KUKA KRL program: ps_b_ltb_res_c02.src, ps_b_ltb_res_c02.dat

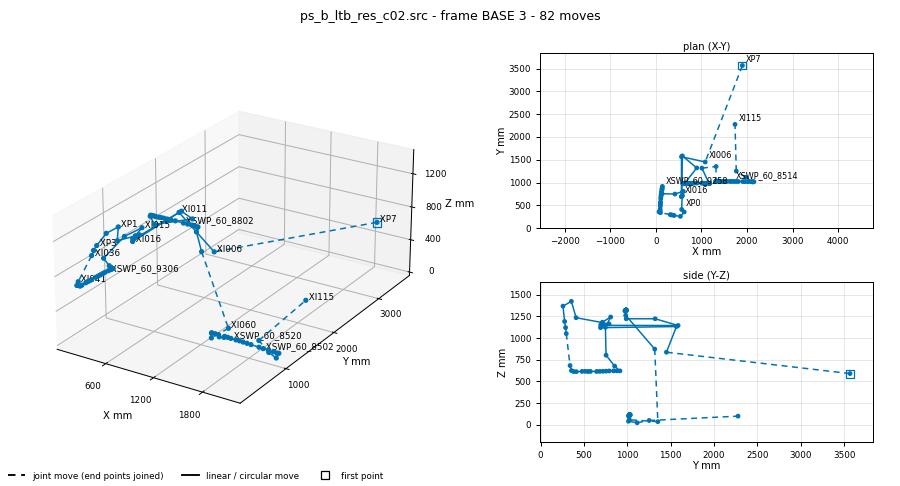
[picture p0: tool path of ps_b_ltb_res_c02.src in frame BASE 3, 82 of 82 moves have a stored position in this frame; points joined in program order, loops and branches not executed]
--- ps_b_ltb_res_c02.src ---
&ACCESS RVO1
&COMMENT Solda Axor LTB
&PARAM DISKPATH = KRC:\R1\Program\OLP
DEF ps_b_ltb_res_c02( )
;FOLD INI
;FOLD SPOTTECH INI
USERSPOT(#INIT)
;ENDFOLD (SPOTTECH INI)
;FOLD GRIPPERTECH INI
USER_GRP(0,DUMMY,DUMMY,GDEFAULT)
;ENDFOLD (GRIPPERTECH INI)
  ;FOLD USER INI
    ;Make your modifications here

  ;ENDFOLD (USER INI)
;ENDFOLD (INI)

; Caracterizacao dos meios de producao
; Changes: Solda Respot - AXOR - LTB
; Versao Atual: 26/03/2016
; Ferramenta : Gun C02
; Name: P13.060-R2

chk_w3_wechs_ok ( )     ; CHECK GUN C2

IF (NOT(GHOST())) THEN
IF MaxStandMenge(3) THEN
  MaxStandmengeErreicht(3)
ENDIF
IF Elektrodenwechsel(3) THEN
  e_Fraes3 ()
ENDIF
ENDIF

;FOLD PTP P7 Vel=100 % PDAT2 Tool[4]:Gun C03 Base[3]:Atego/Axor;%{PE}%R 8.2.20,%MKUKATPBASIS,%CMOVE,%VPTP,%P 1:PTP, 2:P7, 3:, 5:100, 7:PDAT2
$BWDSTART=FALSE
PDAT_ACT=PPDAT2
FDAT_ACT=FP7
BAS(#PTP_PARAMS,100)
PTP XP7
;ENDFOLD

;FOLD OUT 3380 'Perfil Livre Estacao' State=TRUE ;%{PE}%R 8.2.20,%MKUKATPBASIS,%COUT,%VOUTX,%P 2:3380, 3:Perfil Livre Estacao, 5:TRUE, 6:
$OUT[3380]=TRUE
;ENDFOLD
;FOLD WAIT FOR ( IN 3380 'Liberacao de Solda' );%{PE}%R 8.2.20,%MKUKATPBASIS,%CEXT_WAIT_FOR,%VEXT_WAIT_FOR,%P 2:, 4:, 5:$IN, 6:3380, 7:Liberacao de Solda, 9:
WAIT FOR  ( $IN[3380] )
;ENDFOLD
;FOLD OUT 3380 'Perfil Livre Estacao' State=FALSE ;%{PE}%R 8.2.20,%MKUKATPBASIS,%COUT,%VOUTX,%P 2:3380, 3:Perfil Livre Estacao, 5:FALSE, 6:
$OUT[3380]=FALSE
;ENDFOLD

;FOLD ; Liga intertravamento 3 c/ R03;%{PE}%R 8.2.20,%MKUKATPBASIS,%CCOMMENT,%VNORMAL,%P 2:Liga  intertravamento 3 c/  R03
;ENDFOLD
;FOLD Collision.Monitoring_3_On ;%{PE}%MKUKATPUSER
COLLSTOP( 3, 1 ) ;Interrupt-Controlled
;ENDFOLD

;FOLD ; Liga intertravamento 10 c/ R04;%{PE}%R 8.2.20,%MKUKATPBASIS,%CCOMMENT,%VNORMAL,%P 2:Liga  intertravamento 10 c/  R04
;ENDFOLD
;FOLD Collision.Monitoring_10_On ;%{PE}%MKUKATPUSER
COLLSTOP( 10, 1 ) ;not Interrupt-Controlled
;ENDFOLD
;FOLD ; ;%{PE}%R 8.2.20,%MKUKATPBASIS,%CCOMMENT,%VNORMAL,%P 2:
;ENDFOLD
;FOLD ; Liga intertravamento 5 c/ R05;%{PE}%R 8.2.20,%MKUKATPBASIS,%CCOMMENT,%VNORMAL,%P 2:Liga  intertravamento 5 c/  R05
;ENDFOLD
;FOLD Collision.Monitoring_5_On ;%{PE}%MKUKATPUSER
COLLSTOP( 5, 1 ) ;not Interrupt-Controlled
;ENDFOLD

;FOLD ; Liga intertravamento 9 c/ R05;%{PE}%R 8.2.20,%MKUKATPBASIS,%CCOMMENT,%VNORMAL,%P 2:Liga  intertravamento 9 c/  R05
;ENDFOLD
;FOLD Collision.Monitoring_9_On ;%{PE}%MKUKATPUSER
COLLSTOP( 9, 1 ) ;not Interrupt-Controlled
;ENDFOLD

;FOLD ; Liga intertravamento 14 c/ R05;%{PE}%R 8.2.20,%MKUKATPBASIS,%CCOMMENT,%VNORMAL,%P 2:Liga  intertravamento 14 c/  R05
;ENDFOLD
;FOLD Collision.Monitoring_14_On ;%{PE}%MKUKATPUSER
COLLSTOP( 14, 1 ) ;not Interrupt-Controlled
;ENDFOLD
;FOLD ; ;%{PE}%R 8.2.20,%MKUKATPBASIS,%CCOMMENT,%VNORMAL,%P 2:
;ENDFOLD
;FOLD PTP l006 CONT Vel=100 % P_OLP4 Tool[3]:Pinca C2 Base[3]:Atego/Axor;%{PE}%R 8.2.20,%MKUKATPBASIS,%CMOVE,%VPTP,%P 1:PTP, 2:l006, 3:C_DIS, 5:100, 7:P_OLP4
$BWDSTART=FALSE
PDAT_ACT=PP_OLP4
FDAT_ACT=Fl006
BAS(#PTP_PARAMS,100)
PTP Xl006 C_DIS
;ENDFOLD
;FOLD LIN l011 CONT Vel=2 m/s L_OLP48 Tool[3]:Pinca C2 Base[3]:Atego/Axor;%{PE}%R 8.2.20,%MKUKATPBASIS,%CMOVE,%VLIN,%P 1:LIN, 2:l011, 3:C_DIS C_DIS, 5:2, 7:L_OLP48
$BWDSTART=FALSE
LDAT_ACT=LL_OLP48
FDAT_ACT=Fl011
BAS(#CP_PARAMS,2)
LIN Xl011 C_DIS C_DIS
;ENDFOLD
;FOLD LIN l016 CONT Vel=2 m/s L_OLP49 Tool[3]:Pinca C2 Base[3]:Atego/Axor;%{PE}%R 8.2.20,%MKUKATPBASIS,%CMOVE,%VLIN,%P 1:LIN, 2:l016, 3:C_DIS C_DIS, 5:2, 7:L_OLP49
$BWDSTART=FALSE
LDAT_ACT=LL_OLP49
FDAT_ACT=Fl016
BAS(#CP_PARAMS,2)
LIN Xl016 C_DIS C_DIS
;ENDFOLD
;FOLD PTP l021 CONT Vel=100 % P_OLP5 Tool[3]:Pinca C2 Base[3]:Atego/Axor;%{PE}%R 8.2.20,%MKUKATPBASIS,%CMOVE,%VPTP,%P 1:PTP, 2:l021, 3:C_DIS, 5:100, 7:P_OLP5
$BWDSTART=FALSE
PDAT_ACT=PP_OLP5
FDAT_ACT=Fl021
BAS(#PTP_PARAMS,100)
PTP Xl021 C_DIS
;ENDFOLD
;FOLD LIN l026 CONT Vel=2 m/s L_OLP50 Tool[3]:Pinca C2 Base[3]:Atego/Axor;%{PE}%R 8.2.20,%MKUKATPBASIS,%CMOVE,%VLIN,%P 1:LIN, 2:l026, 3:C_DIS C_DIS, 5:2, 7:L_OLP50
$BWDSTART=FALSE
LDAT_ACT=LL_OLP50
FDAT_ACT=Fl026
BAS(#CP_PARAMS,2)
LIN Xl026 C_DIS C_DIS
;ENDFOLD
;FOLD LIN P0 CONT Vel=2 m/s CPDAT0 Tool[3]:Pinca C2 Base[3]:Atego/Axor;%{PE}%R 8.2.20,%MKUKATPBASIS,%CMOVE,%VLIN,%P 1:LIN, 2:P0, 3:C_DIS C_DIS, 5:2, 7:CPDAT0
$BWDSTART=FALSE
LDAT_ACT=LCPDAT0
FDAT_ACT=FP0
BAS(#CP_PARAMS,2)
LIN XP0 C_DIS C_DIS
;ENDFOLD
;FOLD LIN P1 CONT Vel=2 m/s CPDAT1 Tool[3]:Pinca C2 Base[3]:Atego/Axor;%{PE}%R 8.2.20,%MKUKATPBASIS,%CMOVE,%VLIN,%P 1:LIN, 2:P1, 3:C_DIS C_DIS, 5:2, 7:CPDAT1
$BWDSTART=FALSE
LDAT_ACT=LCPDAT1
FDAT_ACT=FP1
BAS(#CP_PARAMS,2)
LIN XP1 C_DIS C_DIS
;ENDFOLD
;FOLD LIN P2 CONT Vel=2 m/s CPDAT2 Tool[3]:Pinca C2 Base[3]:Atego/Axor;%{PE}%R 8.2.20,%MKUKATPBASIS,%CMOVE,%VLIN,%P 1:LIN, 2:P2, 3:C_DIS C_DIS, 5:2, 7:CPDAT2
$BWDSTART=FALSE
LDAT_ACT=LCPDAT2
FDAT_ACT=FP2
BAS(#CP_PARAMS,2)
LIN XP2 C_DIS C_DIS
;ENDFOLD
;FOLD LIN P3 CONT Vel=2 m/s CPDAT3 Tool[3]:Pinca C2 Base[3]:Atego/Axor;%{PE}%R 8.2.20,%MKUKATPBASIS,%CMOVE,%VLIN,%P 1:LIN, 2:P3, 3:C_DIS C_DIS, 5:2, 7:CPDAT3
$BWDSTART=FALSE
LDAT_ACT=LCPDAT3
FDAT_ACT=FP3
BAS(#CP_PARAMS,2)
LIN XP3 C_DIS C_DIS
;ENDFOLD
;FOLD LIN l031 CONT Vel=2 m/s L_OLP51 Tool[3]:Pinca C2 Base[3]:Atego/Axor;%{PE}%R 8.2.20,%MKUKATPBASIS,%CMOVE,%VLIN,%P 1:LIN, 2:l031, 3:C_DIS C_DIS, 5:2, 7:L_OLP51
$BWDSTART=FALSE
LDAT_ACT=LL_OLP51
FDAT_ACT=Fl031
BAS(#CP_PARAMS,2)
LIN Xl031 C_DIS C_DIS
;ENDFOLD
;FOLD PTP l036 CONT Vel=100 % P_OLP6 Tool[3]:Pinca C2 Base[3]:Atego/Axor;%{PE}%R 8.2.20,%MKUKATPBASIS,%CMOVE,%VPTP,%P 1:PTP, 2:l036, 3:C_DIS, 5:100, 7:P_OLP6
$BWDSTART=FALSE
PDAT_ACT=PP_OLP6
FDAT_ACT=Fl036
BAS(#PTP_PARAMS,100)
PTP Xl036 C_DIS
;ENDFOLD
;FOLD PTP l041 CONT Vel=100 % P_OLP7 Tool[3]:Pinca C2 Base[3]:Atego/Axor;%{PE}%R 8.2.20,%MKUKATPBASIS,%CMOVE,%VPTP,%P 1:PTP, 2:l041, 3:C_DIS, 5:100, 7:P_OLP7
$BWDSTART=FALSE
PDAT_ACT=PP_OLP7
FDAT_ACT=Fl041
BAS(#PTP_PARAMS,100)
PTP Xl041 C_DIS
;ENDFOLD
;FOLD LIN l046 CONT Vel=2 m/s L_OLP52 Tool[3]:Pinca C2 Base[3]:Atego/Axor;%{PE}%R 8.2.20,%MKUKATPBASIS,%CMOVE,%VLIN,%P 1:LIN, 2:l046, 3:C_DIS C_DIS, 5:2, 7:L_OLP52
$BWDSTART=FALSE
LDAT_ACT=LL_OLP52
FDAT_ACT=Fl046
BAS(#CP_PARAMS,2)
LIN Xl046 C_DIS C_DIS
;ENDFOLD

;FOLD ; SWP_60_9280;%{PE}%R 8.2.20,%MKUKATPBASIS,%CCOMMENT,%VNORMAL,%P 2:SWP_60_9280
;ENDFOLD
;FOLD LIN SWP_60_9280 L_OLP53 SPOT Gun=2 RETR CLS PgNo1=186 ACTIVE=1 NORMAL Tool[3]:Pinca C2 Base[3]:Atego/Axor;%{PE}%R 8.2.2,%MKUKATPSPOT,%CSPOT,%VLIN,%P 1:LIN, 2:SWP_60_9280, 3:, 5:2, 7:L_OLP53, 10:2, 12:#FIRST, 14:#CLO, 16:186, 18:1, 20:0, 22:0, 24:1, 25:NORMAL
$BWDSTART=FALSE
LDAT_ACT=LL_OLP53
FDAT_ACT=FSWP_60_9280
BAS(#CP_PARAMS,LL_OLP53.VEL)
S_ACT.GUN=2
S_ACT.PAIR=SDEFAULT.PAIR
S_ACT.RETR=#CLO
S_ACT.CLO_TM=1
S_ACT.PGNO1=186
S_ACT.PGNO2=SDEFAULT.PGNO2
S_ACT.PRESS1=SDEFAULT.PRESS1
S_ACT.PRESS2=SDEFAULT.PRESS2
S_READY=FALSE
LIN XSWP_60_9280
USERSPOT(#SPOT, S_ACT)
WAIT FOR S_READY
;ENDFOLD

;FOLD ; SWP_60_9282;%{PE}%R 8.2.20,%MKUKATPBASIS,%CCOMMENT,%VNORMAL,%P 2:SWP_60_9282
;ENDFOLD
;FOLD LIN SWP_60_9282 L_OLP54 SPOT Gun=2 RETR CLS PgNo1=186 ACTIVE=1 NORMAL Tool[3]:Pinca C2 Base[3]:Atego/Axor;%{PE}%R 8.2.2,%MKUKATPSPOT,%CSPOT,%VLIN,%P 1:LIN, 2:SWP_60_9282, 3:, 5:2, 7:L_OLP54, 10:2, 12:#FIRST, 14:#CLO, 16:186, 18:1, 20:0, 22:0, 24:1, 25:NORMAL
$BWDSTART=FALSE
LDAT_ACT=LL_OLP54
FDAT_ACT=FSWP_60_9282
BAS(#CP_PARAMS,LL_OLP54.VEL)
S_ACT.GUN=2
S_ACT.PAIR=SDEFAULT.PAIR
S_ACT.RETR=#CLO
S_ACT.CLO_TM=1
S_ACT.PGNO1=186
S_ACT.PGNO2=SDEFAULT.PGNO2
S_ACT.PRESS1=SDEFAULT.PRESS1
S_ACT.PRESS2=SDEFAULT.PRESS2
S_READY=FALSE
LIN XSWP_60_9282
USERSPOT(#SPOT, S_ACT)
WAIT FOR S_READY
;ENDFOLD

;FOLD ; SWP_60_9286;%{PE}%R 8.2.20,%MKUKATPBASIS,%CCOMMENT,%VNORMAL,%P 2:SWP_60_9286
;ENDFOLD
;FOLD LIN SWP_60_9286 L_OLP55 SPOT Gun=2 RETR CLS PgNo1=186 ACTIVE=1 NORMAL Tool[3]:Pinca C2 Base[3]:Atego/Axor;%{PE}%R 8.2.2,%MKUKATPSPOT,%CSPOT,%VLIN,%P 1:LIN, 2:SWP_60_9286, 3:, 5:2, 7:L_OLP55, 10:2, 12:#FIRST, 14:#CLO, 16:186, 18:1, 20:0, 22:0, 24:1, 25:NORMAL
$BWDSTART=FALSE
LDAT_ACT=LL_OLP55
FDAT_ACT=FSWP_60_9286
BAS(#CP_PARAMS,LL_OLP55.VEL)
S_ACT.GUN=2
S_ACT.PAIR=SDEFAULT.PAIR
S_ACT.RETR=#CLO
S_ACT.CLO_TM=1
S_ACT.PGNO1=186
S_ACT.PGNO2=SDEFAULT.PGNO2
S_ACT.PRESS1=SDEFAULT.PRESS1
S_ACT.PRESS2=SDEFAULT.PRESS2
S_READY=FALSE
LIN XSWP_60_9286
USERSPOT(#SPOT, S_ACT)
WAIT FOR S_READY
;ENDFOLD

;FOLD ; SWP_60_9288;%{PE}%R 8.2.20,%MKUKATPBASIS,%CCOMMENT,%VNORMAL,%P 2:SWP_60_9288
;ENDFOLD
;FOLD LIN SWP_60_9288 L_OLP56 SPOT Gun=2 RETR CLS PgNo1=186 ACTIVE=1 NORMAL Tool[3]:Pinca C2 Base[3]:Atego/Axor;%{PE}%R 8.2.2,%MKUKATPSPOT,%CSPOT,%VLIN,%P 1:LIN, 2:SWP_60_9288, 3:, 5:2, 7:L_OLP56, 10:2, 12:#FIRST, 14:#CLO, 16:186, 18:1, 20:0, 22:0, 24:1, 25:NORMAL
$BWDSTART=FALSE
LDAT_ACT=LL_OLP56
FDAT_ACT=FSWP_60_9288
BAS(#CP_PARAMS,LL_OLP56.VEL)
S_ACT.GUN=2
S_ACT.PAIR=SDEFAULT.PAIR
S_ACT.RETR=#CLO
S_ACT.CLO_TM=1
S_ACT.PGNO1=186
S_ACT.PGNO2=SDEFAULT.PGNO2
S_ACT.PRESS1=SDEFAULT.PRESS1
S_ACT.PRESS2=SDEFAULT.PRESS2
S_READY=FALSE
LIN XSWP_60_9288
USERSPOT(#SPOT, S_ACT)
WAIT FOR S_READY
;ENDFOLD

;FOLD ; SWP_60_9290;%{PE}%R 8.2.20,%MKUKATPBASIS,%CCOMMENT,%VNORMAL,%P 2:SWP_60_9290
;ENDFOLD
;FOLD LIN SWP_60_9290 L_OLP57 SPOT Gun=2 RETR CLS PgNo1=186 ACTIVE=1 NORMAL Tool[3]:Pinca C2 Base[3]:Atego/Axor;%{PE}%R 8.2.2,%MKUKATPSPOT,%CSPOT,%VLIN,%P 1:LIN, 2:SWP_60_9290, 3:, 5:2, 7:L_OLP57, 10:2, 12:#FIRST, 14:#CLO, 16:186, 18:1, 20:0, 22:0, 24:1, 25:NORMAL
$BWDSTART=FALSE
LDAT_ACT=LL_OLP57
FDAT_ACT=FSWP_60_9290
BAS(#CP_PARAMS,LL_OLP57.VEL)
S_ACT.GUN=2
S_ACT.PAIR=SDEFAULT.PAIR
S_ACT.RETR=#CLO
S_ACT.CLO_TM=1
S_ACT.PGNO1=186
S_ACT.PGNO2=SDEFAULT.PGNO2
S_ACT.PRESS1=SDEFAULT.PRESS1
S_ACT.PRESS2=SDEFAULT.PRESS2
S_READY=FALSE
LIN XSWP_60_9290
USERSPOT(#SPOT, S_ACT)
WAIT FOR S_READY
;ENDFOLD

;FOLD ; SWP_60_9292;%{PE}%R 8.2.20,%MKUKATPBASIS,%CCOMMENT,%VNORMAL,%P 2:SWP_60_9292
;ENDFOLD
;FOLD LIN SWP_60_9292 L_OLP58 SPOT Gun=2 RETR CLS PgNo1=186 ACTIVE=1 NORMAL Tool[3]:Pinca C2 Base[3]:Atego/Axor;%{PE}%R 8.2.2,%MKUKATPSPOT,%CSPOT,%VLIN,%P 1:LIN, 2:SWP_60_9292, 3:, 5:2, 7:L_OLP58, 10:2, 12:#FIRST, 14:#CLO, 16:186, 18:1, 20:0, 22:0, 24:1, 25:NORMAL
$BWDSTART=FALSE
LDAT_ACT=LL_OLP58
FDAT_ACT=FSWP_60_9292
BAS(#CP_PARAMS,LL_OLP58.VEL)
S_ACT.GUN=2
S_ACT.PAIR=SDEFAULT.PAIR
S_ACT.RETR=#CLO
S_ACT.CLO_TM=1
S_ACT.PGNO1=186
S_ACT.PGNO2=SDEFAULT.PGNO2
S_ACT.PRESS1=SDEFAULT.PRESS1
S_ACT.PRESS2=SDEFAULT.PRESS2
S_READY=FALSE
LIN XSWP_60_9292
USERSPOT(#SPOT, S_ACT)
WAIT FOR S_READY
;ENDFOLD

;FOLD ; SWP_60_9296;%{PE}%R 8.2.20,%MKUKATPBASIS,%CCOMMENT,%VNORMAL,%P 2:SWP_60_9296
;ENDFOLD
;FOLD LIN SWP_60_9296 L_OLP59 SPOT Gun=2 RETR CLS PgNo1=186 ACTIVE=1 NORMAL Tool[3]:Pinca C2 Base[3]:Atego/Axor;%{PE}%R 8.2.2,%MKUKATPSPOT,%CSPOT,%VLIN,%P 1:LIN, 2:SWP_60_9296, 3:, 5:2, 7:L_OLP59, 10:2, 12:#FIRST, 14:#CLO, 16:186, 18:1, 20:0, 22:0, 24:1, 25:NORMAL
$BWDSTART=FALSE
LDAT_ACT=LL_OLP59
FDAT_ACT=FSWP_60_9296
BAS(#CP_PARAMS,LL_OLP59.VEL)
S_ACT.GUN=2
S_ACT.PAIR=SDEFAULT.PAIR
S_ACT.RETR=#CLO
S_ACT.CLO_TM=1
S_ACT.PGNO1=186
S_ACT.PGNO2=SDEFAULT.PGNO2
S_ACT.PRESS1=SDEFAULT.PRESS1
S_ACT.PRESS2=SDEFAULT.PRESS2
S_READY=FALSE
LIN XSWP_60_9296
USERSPOT(#SPOT, S_ACT)
WAIT FOR S_READY
;ENDFOLD

;FOLD ; SWP_60_9298;%{PE}%R 8.2.20,%MKUKATPBASIS,%CCOMMENT,%VNORMAL,%P 2:SWP_60_9298
;ENDFOLD
;FOLD LIN SWP_60_9298 L_OLP77 SPOT Gun=2 RETR CLS PgNo1=186 ACTIVE=1 NORMAL Tool[3]:Pinca C2 Base[3]:Atego/Axor;%{PE}%R 8.2.2,%MKUKATPSPOT,%CSPOT,%VLIN,%P 1:LIN, 2:SWP_60_9298, 3:, 5:2, 7:L_OLP77, 10:2, 12:#FIRST, 14:#CLO, 16:186, 18:1, 20:0, 22:0, 24:1, 25:NORMAL
$BWDSTART=FALSE
LDAT_ACT=LL_OLP77
FDAT_ACT=FSWP_60_9298
BAS(#CP_PARAMS,LL_OLP77.VEL)
S_ACT.GUN=2
S_ACT.PAIR=SDEFAULT.PAIR
S_ACT.RETR=#CLO
S_ACT.CLO_TM=1
S_ACT.PGNO1=186
S_ACT.PGNO2=SDEFAULT.PGNO2
S_ACT.PRESS1=SDEFAULT.PRESS1
S_ACT.PRESS2=SDEFAULT.PRESS2
S_READY=FALSE
LIN XSWP_60_9298
USERSPOT(#SPOT, S_ACT)
WAIT FOR S_READY
;ENDFOLD

;FOLD ; SWP_60_9300;%{PE}%R 8.2.20,%MKUKATPBASIS,%CCOMMENT,%VNORMAL,%P 2:SWP_60_9300
;ENDFOLD
;FOLD LIN SWP_60_9300 L_OLP78 SPOT Gun=2 RETR CLS PgNo1=186 ACTIVE=1 NORMAL Tool[3]:Pinca C2 Base[3]:Atego/Axor;%{PE}%R 8.2.2,%MKUKATPSPOT,%CSPOT,%VLIN,%P 1:LIN, 2:SWP_60_9300, 3:, 5:2, 7:L_OLP78, 10:2, 12:#FIRST, 14:#CLO, 16:186, 18:1, 20:0, 22:0, 24:1, 25:NORMAL
$BWDSTART=FALSE
LDAT_ACT=LL_OLP78
FDAT_ACT=FSWP_60_9300
BAS(#CP_PARAMS,LL_OLP78.VEL)
S_ACT.GUN=2
S_ACT.PAIR=SDEFAULT.PAIR
S_ACT.RETR=#CLO
S_ACT.CLO_TM=1
S_ACT.PGNO1=186
S_ACT.PGNO2=SDEFAULT.PGNO2
S_ACT.PRESS1=SDEFAULT.PRESS1
S_ACT.PRESS2=SDEFAULT.PRESS2
S_READY=FALSE
LIN XSWP_60_9300
USERSPOT(#SPOT, S_ACT)
WAIT FOR S_READY
;ENDFOLD

;FOLD ; SWP_60_9302;%{PE}%R 8.2.20,%MKUKATPBASIS,%CCOMMENT,%VNORMAL,%P 2:SWP_60_9302
;ENDFOLD
;FOLD LIN SWP_60_9302 L_OLP79 SPOT Gun=2 RETR CLS PgNo1=186 ACTIVE=1 NORMAL Tool[3]:Pinca C2 Base[3]:Atego/Axor;%{PE}%R 8.2.2,%MKUKATPSPOT,%CSPOT,%VLIN,%P 1:LIN, 2:SWP_60_9302, 3:, 5:2, 7:L_OLP79, 10:2, 12:#FIRST, 14:#CLO, 16:186, 18:1, 20:0, 22:0, 24:1, 25:NORMAL
$BWDSTART=FALSE
LDAT_ACT=LL_OLP79
FDAT_ACT=FSWP_60_9302
BAS(#CP_PARAMS,LL_OLP79.VEL)
S_ACT.GUN=2
S_ACT.PAIR=SDEFAULT.PAIR
S_ACT.RETR=#CLO
S_ACT.CLO_TM=1
S_ACT.PGNO1=186
S_ACT.PGNO2=SDEFAULT.PGNO2
S_ACT.PRESS1=SDEFAULT.PRESS1
S_ACT.PRESS2=SDEFAULT.PRESS2
S_READY=FALSE
LIN XSWP_60_9302
USERSPOT(#SPOT, S_ACT)
WAIT FOR S_READY
;ENDFOLD

;FOLD ; SWP_60_9304;%{PE}%R 8.2.20,%MKUKATPBASIS,%CCOMMENT,%VNORMAL,%P 2:SWP_60_9304
;ENDFOLD
;FOLD LIN SWP_60_9304 L_OLP80 SPOT Gun=2 RETR CLS PgNo1=186 ACTIVE=1 NORMAL Tool[3]:Pinca C2 Base[3]:Atego/Axor;%{PE}%R 8.2.2,%MKUKATPSPOT,%CSPOT,%VLIN,%P 1:LIN, 2:SWP_60_9304, 3:, 5:2, 7:L_OLP80, 10:2, 12:#FIRST, 14:#CLO, 16:186, 18:1, 20:0, 22:0, 24:1, 25:NORMAL
$BWDSTART=FALSE
LDAT_ACT=LL_OLP80
FDAT_ACT=FSWP_60_9304
BAS(#CP_PARAMS,LL_OLP80.VEL)
S_ACT.GUN=2
S_ACT.PAIR=SDEFAULT.PAIR
S_ACT.RETR=#CLO
S_ACT.CLO_TM=1
S_ACT.PGNO1=186
S_ACT.PGNO2=SDEFAULT.PGNO2
S_ACT.PRESS1=SDEFAULT.PRESS1
S_ACT.PRESS2=SDEFAULT.PRESS2
S_READY=FALSE
LIN XSWP_60_9304
USERSPOT(#SPOT, S_ACT)
WAIT FOR S_READY
;ENDFOLD

;FOLD ; SWP_60_9306;%{PE}%R 8.2.20,%MKUKATPBASIS,%CCOMMENT,%VNORMAL,%P 2:SWP_60_9306
;ENDFOLD
;FOLD LIN SWP_60_9306 L_OLP81 SPOT Gun=2 RETR CLS PgNo1=186 ACTIVE=1 NORMAL Tool[3]:Pinca C2 Base[3]:Atego/Axor;%{PE}%R 8.2.2,%MKUKATPSPOT,%CSPOT,%VLIN,%P 1:LIN, 2:SWP_60_9306, 3:, 5:2, 7:L_OLP81, 10:2, 12:#FIRST, 14:#CLO, 16:186, 18:1, 20:0, 22:0, 24:1, 25:NORMAL
$BWDSTART=FALSE
LDAT_ACT=LL_OLP81
FDAT_ACT=FSWP_60_9306
BAS(#CP_PARAMS,LL_OLP81.VEL)
S_ACT.GUN=2
S_ACT.PAIR=SDEFAULT.PAIR
S_ACT.RETR=#CLO
S_ACT.CLO_TM=1
S_ACT.PGNO1=186
S_ACT.PGNO2=SDEFAULT.PGNO2
S_ACT.PRESS1=SDEFAULT.PRESS1
S_ACT.PRESS2=SDEFAULT.PRESS2
S_READY=FALSE
LIN XSWP_60_9306
USERSPOT(#SPOT, S_ACT)
WAIT FOR S_READY
;ENDFOLD

;FOLD ; SWP_60_9322;%{PE}%R 8.2.20,%MKUKATPBASIS,%CCOMMENT,%VNORMAL,%P 2:SWP_60_9322
;ENDFOLD
;FOLD LIN SWP_60_9322 L_OLP82 SPOT Gun=2 RETR CLS PgNo1=186 ACTIVE=1 NORMAL Tool[3]:Pinca C2 Base[3]:Atego/Axor;%{PE}%R 8.2.2,%MKUKATPSPOT,%CSPOT,%VLIN,%P 1:LIN, 2:SWP_60_9322, 3:, 5:2, 7:L_OLP82, 10:2, 12:#FIRST, 14:#CLO, 16:186, 18:1, 20:0, 22:0, 24:1, 25:NORMAL
$BWDSTART=FALSE
LDAT_ACT=LL_OLP82
FDAT_ACT=FSWP_60_9322
BAS(#CP_PARAMS,LL_OLP82.VEL)
S_ACT.GUN=2
S_ACT.PAIR=SDEFAULT.PAIR
S_ACT.RETR=#CLO
S_ACT.CLO_TM=1
S_ACT.PGNO1=186
S_ACT.PGNO2=SDEFAULT.PGNO2
S_ACT.PRESS1=SDEFAULT.PRESS1
S_ACT.PRESS2=SDEFAULT.PRESS2
S_READY=FALSE
LIN XSWP_60_9322
USERSPOT(#SPOT, S_ACT)
WAIT FOR S_READY
;ENDFOLD

;FOLD ; SWP_60_9258;%{PE}%R 8.2.20,%MKUKATPBASIS,%CCOMMENT,%VNORMAL,%P 2:SWP_60_9258
;ENDFOLD
;FOLD LIN SWP_60_9258 CPDAT6 SPOT Gun=2 RETR OPN PgNo1=186 ACTIVE=1 NORMAL Tool[3]:Pinca C2 Base[3]:Atego/Axor;%{PE}%R 8.2.2,%MKUKATPSPOT,%CSPOT,%VLIN,%P 1:LIN, 2:SWP_60_9258, 3:, 5:0.001, 7:CPDAT6, 10:2, 12:#FIRST, 14:#OPN, 16:186, 18:1, 20:0, 22:0, 24:1, 25:NORMAL
$BWDSTART=FALSE
LDAT_ACT=LCPDAT6
FDAT_ACT=FSWP_60_9258
BAS(#CP_PARAMS,LCPDAT6.VEL)
S_ACT.GUN=2
S_ACT.PAIR=SDEFAULT.PAIR
S_ACT.RETR=#OPN
S_ACT.CLO_TM=1
S_ACT.PGNO1=186
S_ACT.PGNO2=SDEFAULT.PGNO2
S_ACT.PRESS1=SDEFAULT.PRESS1
S_ACT.PRESS2=SDEFAULT.PRESS2
S_READY=FALSE
LIN XSWP_60_9258
USERSPOT(#SPOT, S_ACT)
WAIT FOR S_READY
;ENDFOLD

;FOLD LIN l051 CONT Vel=1.5 m/s CPDAT8 Tool[3]:Pinca C2 Base[3]:Atego/Axor;%{PE}%R 8.2.20,%MKUKATPBASIS,%CMOVE,%VLIN,%P 1:LIN, 2:l051, 3:C_DIS C_DIS, 5:1.5, 7:CPDAT8
$BWDSTART=FALSE
LDAT_ACT=LCPDAT8
FDAT_ACT=Fl051
BAS(#CP_PARAMS,1.5)
LIN Xl051 C_DIS C_DIS
;ENDFOLD
;FOLD LIN l010 CONT Vel=2 m/s L_OLP2 Tool[3]:Pinca C2 Base[3]:Atego/Axor;%{PE}%R 8.2.20,%MKUKATPBASIS,%CMOVE,%VLIN,%P 1:LIN, 2:l010, 3:C_DIS C_DIS, 5:2, 7:L_OLP2
$BWDSTART=FALSE
LDAT_ACT=LL_OLP2
FDAT_ACT=Fl010
BAS(#CP_PARAMS,2)
LIN Xl010 C_DIS C_DIS
;ENDFOLD
;FOLD LIN P5 CONT Vel=2 m/s CPDAT5 Tool[3]:Pinca C2 Base[3]:Atego/Axor;%{PE}%R 8.2.20,%MKUKATPBASIS,%CMOVE,%VLIN,%P 1:LIN, 2:P5, 3:C_DIS C_DIS, 5:2, 7:CPDAT5
$BWDSTART=FALSE
LDAT_ACT=LCPDAT5
FDAT_ACT=FP5
BAS(#CP_PARAMS,2)
LIN XP5 C_DIS C_DIS
;ENDFOLD
;FOLD LIN l015 CONT Vel=2 m/s L_OLP3 Tool[3]:Pinca C2 Base[3]:Atego/Axor;%{PE}%R 8.2.20,%MKUKATPBASIS,%CMOVE,%VLIN,%P 1:LIN, 2:l015, 3:C_DIS C_DIS, 5:2, 7:L_OLP3
$BWDSTART=FALSE
LDAT_ACT=LL_OLP3
FDAT_ACT=Fl015
BAS(#CP_PARAMS,2)
LIN Xl015 C_DIS C_DIS
;ENDFOLD
;FOLD LIN l020 CONT Vel=2 m/s L_OLP4 Tool[3]:Pinca C2 Base[3]:Atego/Axor;%{PE}%R 8.2.20,%MKUKATPBASIS,%CMOVE,%VLIN,%P 1:LIN, 2:l020, 3:C_DIS C_DIS, 5:2, 7:L_OLP4
$BWDSTART=FALSE
LDAT_ACT=LL_OLP4
FDAT_ACT=Fl020
BAS(#CP_PARAMS,2)
LIN Xl020 C_DIS C_DIS
;ENDFOLD
;FOLD LIN l025 CONT Vel=2 m/s L_OLP5 Tool[3]:Pinca C2 Base[3]:Atego/Axor;%{PE}%R 8.2.20,%MKUKATPBASIS,%CMOVE,%VLIN,%P 1:LIN, 2:l025, 3:C_DIS C_DIS, 5:2, 7:L_OLP5
$BWDSTART=FALSE
LDAT_ACT=LL_OLP5
FDAT_ACT=Fl025
BAS(#CP_PARAMS,2)
LIN Xl025 C_DIS C_DIS
;ENDFOLD
;FOLD LIN l030 CONT Vel=2 m/s L_OLP6 Tool[3]:Pinca C2 Base[3]:Atego/Axor;%{PE}%R 8.2.20,%MKUKATPBASIS,%CMOVE,%VLIN,%P 1:LIN, 2:l030, 3:C_DIS C_DIS, 5:2, 7:L_OLP6
$BWDSTART=FALSE
LDAT_ACT=LL_OLP6
FDAT_ACT=Fl030
BAS(#CP_PARAMS,2)
LIN Xl030 C_DIS C_DIS
;ENDFOLD

;FOLD ; Desliga intertravamento 3 c/ R03;%{PE}%R 8.2.20,%MKUKATPBASIS,%CCOMMENT,%VNORMAL,%P 2:Desliga  intertravamento 3 c/  R03
;ENDFOLD
;FOLD Collision.Monitoring_3_Off . ;%{PE}%MKUKATPUSER
COLLSTOP( 3, 2+0 )
;ENDFOLD

;FOLD ; Desliga intertravamento 10 c/ R04;%{PE}%R 8.2.20,%MKUKATPBASIS,%CCOMMENT,%VNORMAL,%P 2:Desliga  intertravamento 10 c/  R04
;ENDFOLD
;FOLD Collision.Monitoring_10_Off . ;%{PE}%MKUKATPUSER
COLLSTOP( 10, 2+0 )
;ENDFOLD

;FOLD ; Desliga intertravamento 5 c/ R05;%{PE}%R 8.2.20,%MKUKATPBASIS,%CCOMMENT,%VNORMAL,%P 2:Desliga  intertravamento 5 c/  R05
;ENDFOLD
;FOLD Collision.Monitoring_5_Off . ;%{PE}%MKUKATPUSER
COLLSTOP( 5, 2+0 )
;ENDFOLD

;FOLD ; Desliga intertravamento 14 c/ R05;%{PE}%R 8.2.20,%MKUKATPBASIS,%CCOMMENT,%VNORMAL,%P 2:Desliga  intertravamento 14 c/  R05
;ENDFOLD
;FOLD Collision.Monitoring_14_Off . ;%{PE}%MKUKATPUSER
COLLSTOP( 14, 2+0 )
;ENDFOLD

;FOLD LIN l035 CONT Vel=2 m/s L_OLP7 Tool[3]:Pinca C2 Base[3]:Atego/Axor;%{PE}%R 8.2.20,%MKUKATPBASIS,%CMOVE,%VLIN,%P 1:LIN, 2:l035, 3:C_DIS C_DIS, 5:2, 7:L_OLP7
$BWDSTART=FALSE
LDAT_ACT=LL_OLP7
FDAT_ACT=Fl035
BAS(#CP_PARAMS,2)
LIN Xl035 C_DIS C_DIS
;ENDFOLD
;FOLD LIN l040 CONT Vel=2 m/s L_OLP8 Tool[3]:Pinca C2 Base[3]:Atego/Axor;%{PE}%R 8.2.20,%MKUKATPBASIS,%CMOVE,%VLIN,%P 1:LIN, 2:l040, 3:C_DIS C_DIS, 5:2, 7:L_OLP8
$BWDSTART=FALSE
LDAT_ACT=LL_OLP8
FDAT_ACT=Fl040
BAS(#CP_PARAMS,2)
LIN Xl040 C_DIS C_DIS
;ENDFOLD
;FOLD LIN l045 Vel=2 m/s L_OLP9 Tool[3]:Pinca C2 Base[3]:Atego/Axor;%{PE}%R 8.2.20,%MKUKATPBASIS,%CMOVE,%VLIN,%P 1:LIN, 2:l045, 3:, 5:2, 7:L_OLP9
$BWDSTART=FALSE
LDAT_ACT=LL_OLP9
FDAT_ACT=Fl045
BAS(#CP_PARAMS,2)
LIN Xl045
;ENDFOLD

;FOLD ; SWP_60_8580;%{PE}%R 4.1.16,%MKUKATPBASIS,%CCOMMENT,%VNORMAL,%P 2:SWP_60_8580
;ENDFOLD
;FOLD LIN SWP_60_8580 L_OLP10 SPOT Gun=2 RETR CLS PgNo1=183 ACTIVE=1 NORMAL Tool[3]:Pinca C2 Base[3]:Atego/Axor;%{PE}%R 8.2.2,%MKUKATPSPOT,%CSPOT,%VLIN,%P 1:LIN, 2:SWP_60_8580, 3:, 5:2, 7:L_OLP10, 10:2, 12:#FIRST, 14:#CLO, 16:183, 18:1, 20:0, 22:0, 24:1, 25:NORMAL
$BWDSTART=FALSE
LDAT_ACT=LL_OLP10
FDAT_ACT=FSWP_60_8580
BAS(#CP_PARAMS,LL_OLP10.VEL)
S_ACT.GUN=2
S_ACT.PAIR=SDEFAULT.PAIR
S_ACT.RETR=#CLO
S_ACT.CLO_TM=1
S_ACT.PGNO1=183
S_ACT.PGNO2=SDEFAULT.PGNO2
S_ACT.PRESS1=SDEFAULT.PRESS1
S_ACT.PRESS2=SDEFAULT.PRESS2
S_READY=FALSE
LIN XSWP_60_8580
USERSPOT(#SPOT, S_ACT)
WAIT FOR S_READY
;ENDFOLD

;FOLD ; SWP_60_8578;%{PE}%R 4.1.16,%MKUKATPBASIS,%CCOMMENT,%VNORMAL,%P 2:SWP_60_8578
;ENDFOLD
;FOLD LIN SWP_60_8578 L_OLP11 SPOT Gun=2 RETR CLS PgNo1=183 ACTIVE=1 NORMAL Tool[3]:Pinca C2 Base[3]:Atego/Axor;%{PE}%R 8.2.2,%MKUKATPSPOT,%CSPOT,%VLIN,%P 1:LIN, 2:SWP_60_8578, 3:, 5:2, 7:L_OLP11, 10:2, 12:#FIRST, 14:#CLO, 16:183, 18:1, 20:0, 22:0, 24:1, 25:NORMAL
$BWDSTART=FALSE
LDAT_ACT=LL_OLP11
FDAT_ACT=FSWP_60_8578
BAS(#CP_PARAMS,LL_OLP11.VEL)
S_ACT.GUN=2
S_ACT.PAIR=SDEFAULT.PAIR
S_ACT.RETR=#CLO
S_ACT.CLO_TM=1
S_ACT.PGNO1=183
S_ACT.PGNO2=SDEFAULT.PGNO2
S_ACT.PRESS1=SDEFAULT.PRESS1
S_ACT.PRESS2=SDEFAULT.PRESS2
S_READY=FALSE
LIN XSWP_60_8578
USERSPOT(#SPOT, S_ACT)
WAIT FOR S_READY
;ENDFOLD

;FOLD ; SWP_60_8590;%{PE}%R 4.1.16,%MKUKATPBASIS,%CCOMMENT,%VNORMAL,%P 2:SWP_60_8590
;ENDFOLD
;FOLD LIN SWP_60_8590 L_OLP12 SPOT Gun=2 RETR CLS PgNo1=183 ACTIVE=1 NORMAL Tool[3]:Pinca C2 Base[3]:Atego/Axor;%{PE}%R 8.2.2,%MKUKATPSPOT,%CSPOT,%VLIN,%P 1:LIN, 2:SWP_60_8590, 3:, 5:2, 7:L_OLP12, 10:2, 12:#FIRST, 14:#CLO, 16:183, 18:1, 20:0, 22:0, 24:1, 25:NORMAL
$BWDSTART=FALSE
LDAT_ACT=LL_OLP12
FDAT_ACT=FSWP_60_8590
BAS(#CP_PARAMS,LL_OLP12.VEL)
S_ACT.GUN=2
S_ACT.PAIR=SDEFAULT.PAIR
S_ACT.RETR=#CLO
S_ACT.CLO_TM=1
S_ACT.PGNO1=183
S_ACT.PGNO2=SDEFAULT.PGNO2
S_ACT.PRESS1=SDEFAULT.PRESS1
S_ACT.PRESS2=SDEFAULT.PRESS2
S_READY=FALSE
LIN XSWP_60_8590
USERSPOT(#SPOT, S_ACT)
WAIT FOR S_READY
;ENDFOLD

;FOLD LIN l050 CONT Vel=2 m/s L_OLP13 Tool[3]:Pinca C2 Base[3]:Atego/Axor;%{PE}%R 8.2.20,%MKUKATPBASIS,%CMOVE,%VLIN,%P 1:LIN, 2:l050, 3:C_DIS C_DIS, 5:2, 7:L_OLP13
$BWDSTART=FALSE
LDAT_ACT=LL_OLP13
FDAT_ACT=Fl050
BAS(#CP_PARAMS,2)
LIN Xl050 C_DIS C_DIS
;ENDFOLD
;FOLD LIN l023 CONT Vel=0.8 m/s L_OLP83 Tool[3]:Pinca C2 Base[3]:Atego/Axor;%{PE}%R 8.2.20,%MKUKATPBASIS,%CMOVE,%VLIN,%P 1:LIN, 2:l023, 3:C_DIS C_DIS, 5:0.8, 7:L_OLP83
$BWDSTART=FALSE
LDAT_ACT=LL_OLP83
FDAT_ACT=Fl023
BAS(#CP_PARAMS,0.8)
LIN Xl023 C_DIS C_DIS
;ENDFOLD

;FOLD ; SWP_60_8790;%{PE}%R 8.2.20,%MKUKATPBASIS,%CCOMMENT,%VNORMAL,%P 2:SWP_60_8790
;ENDFOLD
;FOLD LIN SWP_60_8790 L_OLP84 SPOT Gun=2 RETR CLS PgNo1=181 ACTIVE=1 NORMAL Tool[3]:Pinca C2 Base[3]:Atego/Axor;%{PE}%R 8.2.2,%MKUKATPSPOT,%CSPOT,%VLIN,%P 1:LIN, 2:SWP_60_8790, 3:, 5:2, 7:L_OLP84, 10:2, 12:#FIRST, 14:#CLO, 16:181, 18:1, 20:0, 22:0, 24:1, 25:NORMAL
$BWDSTART=FALSE
LDAT_ACT=LL_OLP84
FDAT_ACT=FSWP_60_8790
BAS(#CP_PARAMS,LL_OLP84.VEL)
S_ACT.GUN=2
S_ACT.PAIR=SDEFAULT.PAIR
S_ACT.RETR=#CLO
S_ACT.CLO_TM=1
S_ACT.PGNO1=181
S_ACT.PGNO2=SDEFAULT.PGNO2
S_ACT.PRESS1=SDEFAULT.PRESS1
S_ACT.PRESS2=SDEFAULT.PRESS2
S_READY=FALSE
LIN XSWP_60_8790
USERSPOT(#SPOT, S_ACT)
WAIT FOR S_READY
;ENDFOLD

;FOLD ; SWP_60_8792;%{PE}%R 8.2.20,%MKUKATPBASIS,%CCOMMENT,%VNORMAL,%P 2:SWP_60_8792
;ENDFOLD
;FOLD LIN SWP_60_8792 L_OLP85 SPOT Gun=2 RETR CLS PgNo1=181 ACTIVE=1 NORMAL Tool[3]:Pinca C2 Base[3]:Atego/Axor;%{PE}%R 8.2.2,%MKUKATPSPOT,%CSPOT,%VLIN,%P 1:LIN, 2:SWP_60_8792, 3:, 5:2, 7:L_OLP85, 10:2, 12:#FIRST, 14:#CLO, 16:181, 18:1, 20:0, 22:0, 24:1, 25:NORMAL
$BWDSTART=FALSE
LDAT_ACT=LL_OLP85
FDAT_ACT=FSWP_60_8792
BAS(#CP_PARAMS,LL_OLP85.VEL)
S_ACT.GUN=2
S_ACT.PAIR=SDEFAULT.PAIR
S_ACT.RETR=#CLO
S_ACT.CLO_TM=1
S_ACT.PGNO1=181
S_ACT.PGNO2=SDEFAULT.PGNO2
S_ACT.PRESS1=SDEFAULT.PRESS1
S_ACT.PRESS2=SDEFAULT.PRESS2
S_READY=FALSE
LIN XSWP_60_8792
USERSPOT(#SPOT, S_ACT)
WAIT FOR S_READY
;ENDFOLD

;FOLD ; SWP_60_8794;%{PE}%R 8.2.20,%MKUKATPBASIS,%CCOMMENT,%VNORMAL,%P 2:SWP_60_8794
;ENDFOLD
;FOLD LIN SWP_60_8794 L_OLP86 SPOT Gun=2 RETR CLS PgNo1=181 ACTIVE=1 NORMAL Tool[3]:Pinca C2 Base[3]:Atego/Axor;%{PE}%R 8.2.2,%MKUKATPSPOT,%CSPOT,%VLIN,%P 1:LIN, 2:SWP_60_8794, 3:, 5:2, 7:L_OLP86, 10:2, 12:#FIRST, 14:#CLO, 16:181, 18:1, 20:0, 22:0, 24:1, 25:NORMAL
$BWDSTART=FALSE
LDAT_ACT=LL_OLP86
FDAT_ACT=FSWP_60_8794
BAS(#CP_PARAMS,LL_OLP86.VEL)
S_ACT.GUN=2
S_ACT.PAIR=SDEFAULT.PAIR
S_ACT.RETR=#CLO
S_ACT.CLO_TM=1
S_ACT.PGNO1=181
S_ACT.PGNO2=SDEFAULT.PGNO2
S_ACT.PRESS1=SDEFAULT.PRESS1
S_ACT.PRESS2=SDEFAULT.PRESS2
S_READY=FALSE
LIN XSWP_60_8794
USERSPOT(#SPOT, S_ACT)
WAIT FOR S_READY
;ENDFOLD

;FOLD ; SWP_60_8796;%{PE}%R 8.2.20,%MKUKATPBASIS,%CCOMMENT,%VNORMAL,%P 2:SWP_60_8796
;ENDFOLD
;FOLD LIN SWP_60_8796 L_OLP87 SPOT Gun=2 RETR CLS PgNo1=181 ACTIVE=1 NORMAL Tool[3]:Pinca C2 Base[3]:Atego/Axor;%{PE}%R 8.2.2,%MKUKATPSPOT,%CSPOT,%VLIN,%P 1:LIN, 2:SWP_60_8796, 3:, 5:2, 7:L_OLP87, 10:2, 12:#FIRST, 14:#CLO, 16:181, 18:1, 20:0, 22:0, 24:1, 25:NORMAL
$BWDSTART=FALSE
LDAT_ACT=LL_OLP87
FDAT_ACT=FSWP_60_8796
BAS(#CP_PARAMS,LL_OLP87.VEL)
S_ACT.GUN=2
S_ACT.PAIR=SDEFAULT.PAIR
S_ACT.RETR=#CLO
S_ACT.CLO_TM=1
S_ACT.PGNO1=181
S_ACT.PGNO2=SDEFAULT.PGNO2
S_ACT.PRESS1=SDEFAULT.PRESS1
S_ACT.PRESS2=SDEFAULT.PRESS2
S_READY=FALSE
LIN XSWP_60_8796
USERSPOT(#SPOT, S_ACT)
WAIT FOR S_READY
;ENDFOLD

;FOLD ; SWP_60_8798;%{PE}%R 8.2.20,%MKUKATPBASIS,%CCOMMENT,%VNORMAL,%P 2:SWP_60_8798
;ENDFOLD
;FOLD LIN SWP_60_8798 L_OLP88 SPOT Gun=2 RETR CLS PgNo1=181 ACTIVE=1 NORMAL Tool[3]:Pinca C2 Base[3]:Atego/Axor;%{PE}%R 8.2.2,%MKUKATPSPOT,%CSPOT,%VLIN,%P 1:LIN, 2:SWP_60_8798, 3:, 5:2, 7:L_OLP88, 10:2, 12:#FIRST, 14:#CLO, 16:181, 18:1, 20:0, 22:0, 24:1, 25:NORMAL
$BWDSTART=FALSE
LDAT_ACT=LL_OLP88
FDAT_ACT=FSWP_60_8798
BAS(#CP_PARAMS,LL_OLP88.VEL)
S_ACT.GUN=2
S_ACT.PAIR=SDEFAULT.PAIR
S_ACT.RETR=#CLO
S_ACT.CLO_TM=1
S_ACT.PGNO1=181
S_ACT.PGNO2=SDEFAULT.PGNO2
S_ACT.PRESS1=SDEFAULT.PRESS1
S_ACT.PRESS2=SDEFAULT.PRESS2
S_READY=FALSE
LIN XSWP_60_8798
USERSPOT(#SPOT, S_ACT)
WAIT FOR S_READY
;ENDFOLD

;FOLD ; SWP_60_8802;%{PE}%R 8.2.20,%MKUKATPBASIS,%CCOMMENT,%VNORMAL,%P 2:SWP_60_8802
;ENDFOLD
;FOLD LIN SWP_60_8802 L_OLP89 SPOT Gun=2 RETR CLS PgNo1=181 ACTIVE=1 NORMAL Tool[3]:Pinca C2 Base[3]:Atego/Axor;%{PE}%R 8.2.2,%MKUKATPSPOT,%CSPOT,%VLIN,%P 1:LIN, 2:SWP_60_8802, 3:, 5:2, 7:L_OLP89, 10:2, 12:#FIRST, 14:#CLO, 16:181, 18:1, 20:0, 22:0, 24:1, 25:NORMAL
$BWDSTART=FALSE
LDAT_ACT=LL_OLP89
FDAT_ACT=FSWP_60_8802
BAS(#CP_PARAMS,LL_OLP89.VEL)
S_ACT.GUN=2
S_ACT.PAIR=SDEFAULT.PAIR
S_ACT.RETR=#CLO
S_ACT.CLO_TM=1
S_ACT.PGNO1=181
S_ACT.PGNO2=SDEFAULT.PGNO2
S_ACT.PRESS1=SDEFAULT.PRESS1
S_ACT.PRESS2=SDEFAULT.PRESS2
S_READY=FALSE
LIN XSWP_60_8802
USERSPOT(#SPOT, S_ACT)
WAIT FOR S_READY
;ENDFOLD

;FOLD ; SWP_60_8804;%{PE}%R 8.2.20,%MKUKATPBASIS,%CCOMMENT,%VNORMAL,%P 2:SWP_60_8804
;ENDFOLD
;FOLD LIN SWP_60_8804 L_OLP90 SPOT Gun=2 RETR CLS PgNo1=181 ACTIVE=1 NORMAL Tool[3]:Pinca C2 Base[3]:Atego/Axor;%{PE}%R 8.2.2,%MKUKATPSPOT,%CSPOT,%VLIN,%P 1:LIN, 2:SWP_60_8804, 3:, 5:2, 7:L_OLP90, 10:2, 12:#FIRST, 14:#CLO, 16:181, 18:1, 20:0, 22:0, 24:1, 25:NORMAL
$BWDSTART=FALSE
LDAT_ACT=LL_OLP90
FDAT_ACT=FSWP_60_8804
BAS(#CP_PARAMS,LL_OLP90.VEL)
S_ACT.GUN=2
S_ACT.PAIR=SDEFAULT.PAIR
S_ACT.RETR=#CLO
S_ACT.CLO_TM=1
S_ACT.PGNO1=181
S_ACT.PGNO2=SDEFAULT.PGNO2
S_ACT.PRESS1=SDEFAULT.PRESS1
S_ACT.PRESS2=SDEFAULT.PRESS2
S_READY=FALSE
LIN XSWP_60_8804
USERSPOT(#SPOT, S_ACT)
WAIT FOR S_READY
;ENDFOLD

;FOLD ; SWP_60_8806;%{PE}%R 8.2.20,%MKUKATPBASIS,%CCOMMENT,%VNORMAL,%P 2:SWP_60_8806
;ENDFOLD
;FOLD LIN SWP_60_8806 L_OLP91 SPOT Gun=2 RETR CLS PgNo1=181 ACTIVE=1 NORMAL Tool[3]:Pinca C2 Base[3]:Atego/Axor;%{PE}%R 8.2.2,%MKUKATPSPOT,%CSPOT,%VLIN,%P 1:LIN, 2:SWP_60_8806, 3:, 5:2, 7:L_OLP91, 10:2, 12:#FIRST, 14:#CLO, 16:181, 18:1, 20:0, 22:0, 24:1, 25:NORMAL
$BWDSTART=FALSE
LDAT_ACT=LL_OLP91
FDAT_ACT=FSWP_60_8806
BAS(#CP_PARAMS,LL_OLP91.VEL)
S_ACT.GUN=2
S_ACT.PAIR=SDEFAULT.PAIR
S_ACT.RETR=#CLO
S_ACT.CLO_TM=1
S_ACT.PGNO1=181
S_ACT.PGNO2=SDEFAULT.PGNO2
S_ACT.PRESS1=SDEFAULT.PRESS1
S_ACT.PRESS2=SDEFAULT.PRESS2
S_READY=FALSE
LIN XSWP_60_8806
USERSPOT(#SPOT, S_ACT)
WAIT FOR S_READY
;ENDFOLD

;FOLD ; SWP_60_8808;%{PE}%R 8.2.20,%MKUKATPBASIS,%CCOMMENT,%VNORMAL,%P 2:SWP_60_8808
;ENDFOLD
;FOLD LIN SWP_60_8808 L_OLP92 SPOT Gun=2 RETR CLS PgNo1=181 ACTIVE=1 NORMAL Tool[3]:Pinca C2 Base[3]:Atego/Axor;%{PE}%R 8.2.2,%MKUKATPSPOT,%CSPOT,%VLIN,%P 1:LIN, 2:SWP_60_8808, 3:, 5:2, 7:L_OLP92, 10:2, 12:#FIRST, 14:#CLO, 16:181, 18:1, 20:0, 22:0, 24:1, 25:NORMAL
$BWDSTART=FALSE
LDAT_ACT=LL_OLP92
FDAT_ACT=FSWP_60_8808
BAS(#CP_PARAMS,LL_OLP92.VEL)
S_ACT.GUN=2
S_ACT.PAIR=SDEFAULT.PAIR
S_ACT.RETR=#CLO
S_ACT.CLO_TM=1
S_ACT.PGNO1=181
S_ACT.PGNO2=SDEFAULT.PGNO2
S_ACT.PRESS1=SDEFAULT.PRESS1
S_ACT.PRESS2=SDEFAULT.PRESS2
S_READY=FALSE
LIN XSWP_60_8808
USERSPOT(#SPOT, S_ACT)
WAIT FOR S_READY
;ENDFOLD

;FOLD ; SWP_60_8810;%{PE}%R 8.2.20,%MKUKATPBASIS,%CCOMMENT,%VNORMAL,%P 2:SWP_60_8810
;ENDFOLD
;FOLD LIN SWP_60_8810 L_OLP93 SPOT Gun=2 RETR CLS PgNo1=181 ACTIVE=1 NORMAL Tool[3]:Pinca C2 Base[3]:Atego/Axor;%{PE}%R 8.2.2,%MKUKATPSPOT,%CSPOT,%VLIN,%P 1:LIN, 2:SWP_60_8810, 3:, 5:2, 7:L_OLP93, 10:2, 12:#FIRST, 14:#CLO, 16:181, 18:1, 20:0, 22:0, 24:1, 25:NORMAL
$BWDSTART=FALSE
LDAT_ACT=LL_OLP93
FDAT_ACT=FSWP_60_8810
BAS(#CP_PARAMS,LL_OLP93.VEL)
S_ACT.GUN=2
S_ACT.PAIR=SDEFAULT.PAIR
S_ACT.RETR=#CLO
S_ACT.CLO_TM=1
S_ACT.PGNO1=181
S_ACT.PGNO2=SDEFAULT.PGNO2
S_ACT.PRESS1=SDEFAULT.PRESS1
S_ACT.PRESS2=SDEFAULT.PRESS2
S_READY=FALSE
LIN XSWP_60_8810
USERSPOT(#SPOT, S_ACT)
WAIT FOR S_READY
;ENDFOLD

;FOLD LIN l028 Vel=2 m/s L_OLP94 Tool[3]:Pinca C2 Base[3]:Atego/Axor;%{PE}%R 8.2.20,%MKUKATPBASIS,%CMOVE,%VLIN,%P 1:LIN, 2:l028, 3:, 5:2, 7:L_OLP94
$BWDSTART=FALSE
LDAT_ACT=LL_OLP94
FDAT_ACT=Fl028
BAS(#CP_PARAMS,2)
LIN Xl028
;ENDFOLD
;FOLD LIN l033 CONT Vel=2 m/s L_OLP95 Tool[3]:Pinca C2 Base[3]:Atego/Axor;%{PE}%R 8.2.20,%MKUKATPBASIS,%CMOVE,%VLIN,%P 1:LIN, 2:l033, 3:C_DIS C_DIS, 5:2, 7:L_OLP95
$BWDSTART=FALSE
LDAT_ACT=LL_OLP95
FDAT_ACT=Fl033
BAS(#CP_PARAMS,2)
LIN Xl033 C_DIS C_DIS
;ENDFOLD
;FOLD LIN P6 CONT Vel=2 m/s CPDAT7 Tool[3]:Pinca C2 Base[3]:Atego/Axor;%{PE}%R 8.2.20,%MKUKATPBASIS,%CMOVE,%VLIN,%P 1:LIN, 2:P6, 3:C_DIS C_DIS, 5:2, 7:CPDAT7
$BWDSTART=FALSE
LDAT_ACT=LCPDAT7
FDAT_ACT=FP6
BAS(#CP_PARAMS,2)
LIN XP6 C_DIS C_DIS
;ENDFOLD

;FOLD ; Desliga intertravamento 9 c/ R05;%{PE}%R 8.2.20,%MKUKATPBASIS,%CCOMMENT,%VNORMAL,%P 2:Desliga  intertravamento 9 c/  R05
;ENDFOLD
;FOLD Collision.Monitoring_9_Off . ;%{PE}%MKUKATPUSER
COLLSTOP( 9, 2+0 )
;ENDFOLD

;FOLD PTP l060 CONT Vel=100 % PDAT3 Tool[3]:Pinca C2 Base[3]:Atego/Axor;%{PE}%R 8.2.20,%MKUKATPBASIS,%CMOVE,%VPTP,%P 1:PTP, 2:l060, 3:C_DIS, 5:100, 7:PDAT3
$BWDSTART=FALSE
PDAT_ACT=PPDAT3
FDAT_ACT=Fl060
BAS(#PTP_PARAMS,100)
PTP Xl060 C_DIS
;ENDFOLD
;FOLD PTP P10 CONT Vel=100 % PDAT4 Tool[3]:Pinca C2 Base[3]:Atego/Axor;%{PE}%R 8.2.20,%MKUKATPBASIS,%CMOVE,%VPTP,%P 1:PTP, 2:P10, 3:C_DIS, 5:100, 7:PDAT4
$BWDSTART=FALSE
PDAT_ACT=PPDAT4
FDAT_ACT=FP10
BAS(#PTP_PARAMS,100)
PTP XP10 C_DIS
;ENDFOLD
;FOLD LIN l075  Vel=2.00 m/s L_OLP18 Tool[3]:Gun C02 Base[3]:Atego/Axor;%{PE}%R8.2.19,%MKUKATPBASIS,%CMOVE,%VLIN,%P 1:LIN, 2:l075, 3: , 5:2.00, 7:L_OLP18
$BWDSTART = FALSE
LDAT_ACT= LL_OLP18
FDAT_ACT= Fl075
BAS(#CP_PARAMS,2.00)
LIN Xl075
;ENDFOLD

;FOLD ; SWP_60_8532;%{PE}%R 4.1.16,%MKUKATPBASIS,%CCOMMENT,%VNORMAL,%P 2:SWP_60_8532
;ENDFOLD
;FOLD LIN SWP_60_8532 L_OLP19 SPOT Gun=2 RETR CLS PgNo1=187 ACTIVE=1 NORMAL Tool[3]:Pinca C2 Base[3]:Atego/Axor;%{PE}%R 8.2.2,%MKUKATPSPOT,%CSPOT,%VLIN,%P 1:LIN, 2:SWP_60_8532, 3:, 5:2, 7:L_OLP19, 10:2, 12:#FIRST, 14:#CLO, 16:187, 18:1, 20:0, 22:0, 24:1, 25:NORMAL
$BWDSTART=FALSE
LDAT_ACT=LL_OLP19
FDAT_ACT=FSWP_60_8532
BAS(#CP_PARAMS,LL_OLP19.VEL)
S_ACT.GUN=2
S_ACT.PAIR=SDEFAULT.PAIR
S_ACT.RETR=#CLO
S_ACT.CLO_TM=1
S_ACT.PGNO1=187
S_ACT.PGNO2=SDEFAULT.PGNO2
S_ACT.PRESS1=SDEFAULT.PRESS1
S_ACT.PRESS2=SDEFAULT.PRESS2
S_READY=FALSE
LIN XSWP_60_8532
USERSPOT(#SPOT, S_ACT)
WAIT FOR S_READY
;ENDFOLD

;FOLD ; SWP_60_8530;%{PE}%R 4.1.16,%MKUKATPBASIS,%CCOMMENT,%VNORMAL,%P 2:SWP_60_8530
;ENDFOLD
;FOLD LIN SWP_60_8530 L_OLP20 SPOT Gun=2 RETR CLS PgNo1=187 ACTIVE=1 NORMAL Tool[3]:Pinca C2 Base[3]:Atego/Axor;%{PE}%R 8.2.2,%MKUKATPSPOT,%CSPOT,%VLIN,%P 1:LIN, 2:SWP_60_8530, 3:, 5:2, 7:L_OLP20, 10:2, 12:#FIRST, 14:#CLO, 16:187, 18:1, 20:0, 22:0, 24:1, 25:NORMAL
$BWDSTART=FALSE
LDAT_ACT=LL_OLP20
FDAT_ACT=FSWP_60_8530
BAS(#CP_PARAMS,LL_OLP20.VEL)
S_ACT.GUN=2
S_ACT.PAIR=SDEFAULT.PAIR
S_ACT.RETR=#CLO
S_ACT.CLO_TM=1
S_ACT.PGNO1=187
S_ACT.PGNO2=SDEFAULT.PGNO2
S_ACT.PRESS1=SDEFAULT.PRESS1
S_ACT.PRESS2=SDEFAULT.PRESS2
S_READY=FALSE
LIN XSWP_60_8530
USERSPOT(#SPOT, S_ACT)
WAIT FOR S_READY
;ENDFOLD

;FOLD ; SWP_60_8528;%{PE}%R 4.1.16,%MKUKATPBASIS,%CCOMMENT,%VNORMAL,%P 2:SWP_60_8528
;ENDFOLD
;FOLD LIN SWP_60_8528 L_OLP21 SPOT Gun=2 RETR CLS PgNo1=187 ACTIVE=1 NORMAL Tool[3]:Pinca C2 Base[3]:Atego/Axor;%{PE}%R 8.2.2,%MKUKATPSPOT,%CSPOT,%VLIN,%P 1:LIN, 2:SWP_60_8528, 3:, 5:2, 7:L_OLP21, 10:2, 12:#FIRST, 14:#CLO, 16:187, 18:1, 20:0, 22:0, 24:1, 25:NORMAL
$BWDSTART=FALSE
LDAT_ACT=LL_OLP21
FDAT_ACT=FSWP_60_8528
BAS(#CP_PARAMS,LL_OLP21.VEL)
S_ACT.GUN=2
S_ACT.PAIR=SDEFAULT.PAIR
S_ACT.RETR=#CLO
S_ACT.CLO_TM=1
S_ACT.PGNO1=187
S_ACT.PGNO2=SDEFAULT.PGNO2
S_ACT.PRESS1=SDEFAULT.PRESS1
S_ACT.PRESS2=SDEFAULT.PRESS2
S_READY=FALSE
LIN XSWP_60_8528
USERSPOT(#SPOT, S_ACT)
WAIT FOR S_READY
;ENDFOLD

;FOLD LIN l080 CONT Vel=2 m/s L_OLP22 Tool[3]:Pinca C2 Base[3]:Atego/Axor;%{PE}%R 8.2.20,%MKUKATPBASIS,%CMOVE,%VLIN,%P 1:LIN, 2:l080, 3:C_DIS C_DIS, 5:2, 7:L_OLP22
$BWDSTART=FALSE
LDAT_ACT=LL_OLP22
FDAT_ACT=Fl080
BAS(#CP_PARAMS,2)
LIN Xl080 C_DIS C_DIS
;ENDFOLD
;FOLD LIN l085 CONT Vel=2 m/s L_OLP23 Tool[3]:Pinca C2 Base[3]:Atego/Axor;%{PE}%R 8.2.20,%MKUKATPBASIS,%CMOVE,%VLIN,%P 1:LIN, 2:l085, 3:C_DIS C_DIS, 5:2, 7:L_OLP23
$BWDSTART=FALSE
LDAT_ACT=LL_OLP23
FDAT_ACT=Fl085
BAS(#CP_PARAMS,2)
LIN Xl085 C_DIS C_DIS
;ENDFOLD

;FOLD ; SWP_60_8524;%{PE}%R 4.1.16,%MKUKATPBASIS,%CCOMMENT,%VNORMAL,%P 2:SWP_60_8524
;ENDFOLD
;FOLD LIN SWP_60_8524 L_OLP24 SPOT Gun=2 RETR CLS PgNo1=187 ACTIVE=1 NORMAL Tool[3]:Pinca C2 Base[3]:Atego/Axor;%{PE}%R 8.2.2,%MKUKATPSPOT,%CSPOT,%VLIN,%P 1:LIN, 2:SWP_60_8524, 3:, 5:2, 7:L_OLP24, 10:2, 12:#FIRST, 14:#CLO, 16:187, 18:1, 20:0, 22:0, 24:1, 25:NORMAL
$BWDSTART=FALSE
LDAT_ACT=LL_OLP24
FDAT_ACT=FSWP_60_8524
BAS(#CP_PARAMS,LL_OLP24.VEL)
S_ACT.GUN=2
S_ACT.PAIR=SDEFAULT.PAIR
S_ACT.RETR=#CLO
S_ACT.CLO_TM=1
S_ACT.PGNO1=187
S_ACT.PGNO2=SDEFAULT.PGNO2
S_ACT.PRESS1=SDEFAULT.PRESS1
S_ACT.PRESS2=SDEFAULT.PRESS2
S_READY=FALSE
LIN XSWP_60_8524
USERSPOT(#SPOT, S_ACT)
WAIT FOR S_READY
;ENDFOLD

;FOLD ; SWP_60_8522;%{PE}%R 4.1.16,%MKUKATPBASIS,%CCOMMENT,%VNORMAL,%P 2:SWP_60_8522
;ENDFOLD
;FOLD LIN SWP_60_8522 L_OLP25 SPOT Gun=2 RETR CLS PgNo1=187 ACTIVE=1 NORMAL Tool[3]:Pinca C2 Base[3]:Atego/Axor;%{PE}%R 8.2.2,%MKUKATPSPOT,%CSPOT,%VLIN,%P 1:LIN, 2:SWP_60_8522, 3:, 5:2, 7:L_OLP25, 10:2, 12:#FIRST, 14:#CLO, 16:187, 18:1, 20:0, 22:0, 24:1, 25:NORMAL
$BWDSTART=FALSE
LDAT_ACT=LL_OLP25
FDAT_ACT=FSWP_60_8522
BAS(#CP_PARAMS,LL_OLP25.VEL)
S_ACT.GUN=2
S_ACT.PAIR=SDEFAULT.PAIR
S_ACT.RETR=#CLO
S_ACT.CLO_TM=1
S_ACT.PGNO1=187
S_ACT.PGNO2=SDEFAULT.PGNO2
S_ACT.PRESS1=SDEFAULT.PRESS1
S_ACT.PRESS2=SDEFAULT.PRESS2
S_READY=FALSE
LIN XSWP_60_8522
USERSPOT(#SPOT, S_ACT)
WAIT FOR S_READY
;ENDFOLD

;FOLD ; SWP_60_8520;%{PE}%R 4.1.16,%MKUKATPBASIS,%CCOMMENT,%VNORMAL,%P 2:SWP_60_8520
;ENDFOLD
;FOLD LIN SWP_60_8520 L_OLP26 SPOT Gun=2 RETR CLS PgNo1=189 ACTIVE=1 NORMAL Tool[3]:Pinca C2 Base[3]:Atego/Axor;%{PE}%R 8.2.2,%MKUKATPSPOT,%CSPOT,%VLIN,%P 1:LIN, 2:SWP_60_8520, 3:, 5:2, 7:L_OLP26, 10:2, 12:#FIRST, 14:#CLO, 16:189, 18:1, 20:0, 22:0, 24:1, 25:NORMAL
$BWDSTART=FALSE
LDAT_ACT=LL_OLP26
FDAT_ACT=FSWP_60_8520
BAS(#CP_PARAMS,LL_OLP26.VEL)
S_ACT.GUN=2
S_ACT.PAIR=SDEFAULT.PAIR
S_ACT.RETR=#CLO
S_ACT.CLO_TM=1
S_ACT.PGNO1=189
S_ACT.PGNO2=SDEFAULT.PGNO2
S_ACT.PRESS1=SDEFAULT.PRESS1
S_ACT.PRESS2=SDEFAULT.PRESS2
S_READY=FALSE
LIN XSWP_60_8520
USERSPOT(#SPOT, S_ACT)
WAIT FOR S_READY
;ENDFOLD

;FOLD ; SWP_60_8516;%{PE}%R 4.1.16,%MKUKATPBASIS,%CCOMMENT,%VNORMAL,%P 2:SWP_60_8516
;ENDFOLD
;FOLD LIN SWP_60_8516 L_OLP29 SPOT Gun=2 RETR CLS PgNo1=189 ACTIVE=1 NORMAL Tool[3]:Pinca C2 Base[3]:Atego/Axor;%{PE}%R 8.2.2,%MKUKATPSPOT,%CSPOT,%VLIN,%P 1:LIN, 2:SWP_60_8516, 3:, 5:2, 7:L_OLP29, 10:2, 12:#FIRST, 14:#CLO, 16:189, 18:1, 20:0, 22:0, 24:1, 25:NORMAL
$BWDSTART=FALSE
LDAT_ACT=LL_OLP29
FDAT_ACT=FSWP_60_8516
BAS(#CP_PARAMS,LL_OLP29.VEL)
S_ACT.GUN=2
S_ACT.PAIR=SDEFAULT.PAIR
S_ACT.RETR=#CLO
S_ACT.CLO_TM=1
S_ACT.PGNO1=189
S_ACT.PGNO2=SDEFAULT.PGNO2
S_ACT.PRESS1=SDEFAULT.PRESS1
S_ACT.PRESS2=SDEFAULT.PRESS2
S_READY=FALSE
LIN XSWP_60_8516
USERSPOT(#SPOT, S_ACT)
WAIT FOR S_READY
;ENDFOLD

;FOLD ; SWP_60_8514;%{PE}%R 4.1.16,%MKUKATPBASIS,%CCOMMENT,%VNORMAL,%P 2:SWP_60_8514
;ENDFOLD
;FOLD LIN SWP_60_8514 L_OLP30 SPOT Gun=2 RETR CLS PgNo1=185 ACTIVE=1 NORMAL Tool[3]:Pinca C2 Base[3]:Atego/Axor;%{PE}%R 8.2.2,%MKUKATPSPOT,%CSPOT,%VLIN,%P 1:LIN, 2:SWP_60_8514, 3:, 5:2, 7:L_OLP30, 10:2, 12:#FIRST, 14:#CLO, 16:185, 18:1, 20:0, 22:0, 24:1, 25:NORMAL
$BWDSTART=FALSE
LDAT_ACT=LL_OLP30
FDAT_ACT=FSWP_60_8514
BAS(#CP_PARAMS,LL_OLP30.VEL)
S_ACT.GUN=2
S_ACT.PAIR=SDEFAULT.PAIR
S_ACT.RETR=#CLO
S_ACT.CLO_TM=1
S_ACT.PGNO1=185
S_ACT.PGNO2=SDEFAULT.PGNO2
S_ACT.PRESS1=SDEFAULT.PRESS1
S_ACT.PRESS2=SDEFAULT.PRESS2
S_READY=FALSE
LIN XSWP_60_8514
USERSPOT(#SPOT, S_ACT)
WAIT FOR S_READY
;ENDFOLD

;FOLD ; SWP_60_8512;%{PE}%R 4.1.16,%MKUKATPBASIS,%CCOMMENT,%VNORMAL,%P 2:SWP_60_8512
;ENDFOLD
;FOLD LIN SWP_60_8512 L_OLP31 SPOT Gun=2 RETR CLS PgNo1=185 ACTIVE=1 NORMAL Tool[3]:Pinca C2 Base[3]:Atego/Axor;%{PE}%R 8.2.2,%MKUKATPSPOT,%CSPOT,%VLIN,%P 1:LIN, 2:SWP_60_8512, 3:, 5:2, 7:L_OLP31, 10:2, 12:#FIRST, 14:#CLO, 16:185, 18:1, 20:0, 22:0, 24:1, 25:NORMAL
$BWDSTART=FALSE
LDAT_ACT=LL_OLP31
FDAT_ACT=FSWP_60_8512
BAS(#CP_PARAMS,LL_OLP31.VEL)
S_ACT.GUN=2
S_ACT.PAIR=SDEFAULT.PAIR
S_ACT.RETR=#CLO
S_ACT.CLO_TM=1
S_ACT.PGNO1=185
S_ACT.PGNO2=SDEFAULT.PGNO2
S_ACT.PRESS1=SDEFAULT.PRESS1
S_ACT.PRESS2=SDEFAULT.PRESS2
S_READY=FALSE
LIN XSWP_60_8512
USERSPOT(#SPOT, S_ACT)
WAIT FOR S_READY
;ENDFOLD

;FOLD ; SWP_60_8510;%{PE}%R 4.1.16,%MKUKATPBASIS,%CCOMMENT,%VNORMAL,%P 2:SWP_60_8510
;ENDFOLD
;FOLD LIN SWP_60_8510 L_OLP32 SPOT Gun=2 RETR CLS PgNo1=185 ACTIVE=1 NORMAL Tool[3]:Pinca C2 Base[3]:Atego/Axor;%{PE}%R 8.2.2,%MKUKATPSPOT,%CSPOT,%VLIN,%P 1:LIN, 2:SWP_60_8510, 3:, 5:2, 7:L_OLP32, 10:2, 12:#FIRST, 14:#CLO, 16:185, 18:1, 20:0, 22:0, 24:1, 25:NORMAL
$BWDSTART=FALSE
LDAT_ACT=LL_OLP32
FDAT_ACT=FSWP_60_8510
BAS(#CP_PARAMS,LL_OLP32.VEL)
S_ACT.GUN=2
S_ACT.PAIR=SDEFAULT.PAIR
S_ACT.RETR=#CLO
S_ACT.CLO_TM=1
S_ACT.PGNO1=185
S_ACT.PGNO2=SDEFAULT.PGNO2
S_ACT.PRESS1=SDEFAULT.PRESS1
S_ACT.PRESS2=SDEFAULT.PRESS2
S_READY=FALSE
LIN XSWP_60_8510
USERSPOT(#SPOT, S_ACT)
WAIT FOR S_READY
;ENDFOLD

;FOLD ; SWP_60_8508;%{PE}%R 4.1.16,%MKUKATPBASIS,%CCOMMENT,%VNORMAL,%P 2:SWP_60_8508
;ENDFOLD
;FOLD LIN SWP_60_8508 L_OLP33 SPOT Gun=2 RETR CLS PgNo1=187 ACTIVE=1 NORMAL Tool[3]:Pinca C2 Base[3]:Atego/Axor;%{PE}%R 8.2.2,%MKUKATPSPOT,%CSPOT,%VLIN,%P 1:LIN, 2:SWP_60_8508, 3:, 5:2, 7:L_OLP33, 10:2, 12:#FIRST, 14:#CLO, 16:187, 18:1, 20:0, 22:0, 24:1, 25:NORMAL
$BWDSTART=FALSE
LDAT_ACT=LL_OLP33
FDAT_ACT=FSWP_60_8508
BAS(#CP_PARAMS,LL_OLP33.VEL)
S_ACT.GUN=2
S_ACT.PAIR=SDEFAULT.PAIR
S_ACT.RETR=#CLO
S_ACT.CLO_TM=1
S_ACT.PGNO1=187
S_ACT.PGNO2=SDEFAULT.PGNO2
S_ACT.PRESS1=SDEFAULT.PRESS1
S_ACT.PRESS2=SDEFAULT.PRESS2
S_READY=FALSE
LIN XSWP_60_8508
USERSPOT(#SPOT, S_ACT)
WAIT FOR S_READY
;ENDFOLD

;FOLD ; SWP_60_8504;%{PE}%R 4.1.16,%MKUKATPBASIS,%CCOMMENT,%VNORMAL,%P 2:SWP_60_8504
;ENDFOLD
;FOLD LIN SWP_60_8504 L_OLP34 SPOT Gun=2 RETR CLS PgNo1=185 ACTIVE=1 NORMAL Tool[3]:Pinca C2 Base[3]:Atego/Axor;%{PE}%R 8.2.2,%MKUKATPSPOT,%CSPOT,%VLIN,%P 1:LIN, 2:SWP_60_8504, 3:, 5:2, 7:L_OLP34, 10:2, 12:#FIRST, 14:#CLO, 16:185, 18:1, 20:0, 22:0, 24:1, 25:NORMAL
$BWDSTART=FALSE
LDAT_ACT=LL_OLP34
FDAT_ACT=FSWP_60_8504
BAS(#CP_PARAMS,LL_OLP34.VEL)
S_ACT.GUN=2
S_ACT.PAIR=SDEFAULT.PAIR
S_ACT.RETR=#CLO
S_ACT.CLO_TM=1
S_ACT.PGNO1=185
S_ACT.PGNO2=SDEFAULT.PGNO2
S_ACT.PRESS1=SDEFAULT.PRESS1
S_ACT.PRESS2=SDEFAULT.PRESS2
S_READY=FALSE
LIN XSWP_60_8504
USERSPOT(#SPOT, S_ACT)
WAIT FOR S_READY
;ENDFOLD

;FOLD ; SWP_60_8502;%{PE}%R 4.1.16,%MKUKATPBASIS,%CCOMMENT,%VNORMAL,%P 2:SWP_60_8502
;ENDFOLD
;FOLD LIN SWP_60_8502 L_OLP35 SPOT Gun=2 RETR CLS PgNo1=185 ACTIVE=1 NORMAL Tool[3]:Pinca C2 Base[3]:Atego/Axor;%{PE}%R 8.2.2,%MKUKATPSPOT,%CSPOT,%VLIN,%P 1:LIN, 2:SWP_60_8502, 3:, 5:2, 7:L_OLP35, 10:2, 12:#FIRST, 14:#CLO, 16:185, 18:1, 20:0, 22:0, 24:1, 25:NORMAL
$BWDSTART=FALSE
LDAT_ACT=LL_OLP35
FDAT_ACT=FSWP_60_8502
BAS(#CP_PARAMS,LL_OLP35.VEL)
S_ACT.GUN=2
S_ACT.PAIR=SDEFAULT.PAIR
S_ACT.RETR=#CLO
S_ACT.CLO_TM=1
S_ACT.PGNO1=185
S_ACT.PGNO2=SDEFAULT.PGNO2
S_ACT.PRESS1=SDEFAULT.PRESS1
S_ACT.PRESS2=SDEFAULT.PRESS2
S_READY=FALSE
LIN XSWP_60_8502
USERSPOT(#SPOT, S_ACT)
WAIT FOR S_READY
;ENDFOLD

;FOLD ; SWP_60_8500;%{PE}%R 4.1.16,%MKUKATPBASIS,%CCOMMENT,%VNORMAL,%P 2:SWP_60_8500
;ENDFOLD
;FOLD LIN SWP_60_8500 L_OLP36 SPOT Gun=2 RETR CLS PgNo1=185 ACTIVE=1 NORMAL Tool[3]:Pinca C2 Base[3]:Atego/Axor;%{PE}%R 8.2.2,%MKUKATPSPOT,%CSPOT,%VLIN,%P 1:LIN, 2:SWP_60_8500, 3:, 5:2, 7:L_OLP36, 10:2, 12:#FIRST, 14:#CLO, 16:185, 18:1, 20:0, 22:0, 24:1, 25:NORMAL
$BWDSTART=FALSE
LDAT_ACT=LL_OLP36
FDAT_ACT=FSWP_60_8500
BAS(#CP_PARAMS,LL_OLP36.VEL)
S_ACT.GUN=2
S_ACT.PAIR=SDEFAULT.PAIR
S_ACT.RETR=#CLO
S_ACT.CLO_TM=1
S_ACT.PGNO1=185
S_ACT.PGNO2=SDEFAULT.PGNO2
S_ACT.PRESS1=SDEFAULT.PRESS1
S_ACT.PRESS2=SDEFAULT.PRESS2
S_READY=FALSE
LIN XSWP_60_8500
USERSPOT(#SPOT, S_ACT)
WAIT FOR S_READY
;ENDFOLD

;FOLD ; SWP_60_8498;%{PE}%R 4.1.16,%MKUKATPBASIS,%CCOMMENT,%VNORMAL,%P 2:SWP_60_8498
;ENDFOLD
;FOLD LIN SWP_60_8498 L_OLP37 SPOT Gun=2 RETR CLS PgNo1=185 ACTIVE=1 NORMAL Tool[3]:Pinca C2 Base[3]:Atego/Axor;%{PE}%R 8.2.2,%MKUKATPSPOT,%CSPOT,%VLIN,%P 1:LIN, 2:SWP_60_8498, 3:, 5:2, 7:L_OLP37, 10:2, 12:#FIRST, 14:#CLO, 16:185, 18:1, 20:0, 22:0, 24:1, 25:NORMAL
$BWDSTART=FALSE
LDAT_ACT=LL_OLP37
FDAT_ACT=FSWP_60_8498
BAS(#CP_PARAMS,LL_OLP37.VEL)
S_ACT.GUN=2
S_ACT.PAIR=SDEFAULT.PAIR
S_ACT.RETR=#CLO
S_ACT.CLO_TM=1
S_ACT.PGNO1=185
S_ACT.PGNO2=SDEFAULT.PGNO2
S_ACT.PRESS1=SDEFAULT.PRESS1
S_ACT.PRESS2=SDEFAULT.PRESS2
S_READY=FALSE
LIN XSWP_60_8498
USERSPOT(#SPOT, S_ACT)
WAIT FOR S_READY
;ENDFOLD

;FOLD ; SWP_60_8398;%{PE}%R 8.2.20,%MKUKATPBASIS,%CCOMMENT,%VNORMAL,%P 2:SWP_60_8398
;ENDFOLD
;FOLD LIN SWP_60_8398 L_OLP38 SPOT Gun=2 RETR CLS PgNo1=185 ACTIVE=1 NORMAL Tool[3]:Pinca C2 Base[3]:Atego/Axor;%{PE}%R 8.2.2,%MKUKATPSPOT,%CSPOT,%VLIN,%P 1:LIN, 2:SWP_60_8398, 3:, 5:2, 7:L_OLP38, 10:2, 12:#FIRST, 14:#CLO, 16:185, 18:1, 20:0, 22:0, 24:1, 25:NORMAL
$BWDSTART=FALSE
LDAT_ACT=LL_OLP38
FDAT_ACT=FSWP_60_8398
BAS(#CP_PARAMS,LL_OLP38.VEL)
S_ACT.GUN=2
S_ACT.PAIR=SDEFAULT.PAIR
S_ACT.RETR=#CLO
S_ACT.CLO_TM=1
S_ACT.PGNO1=185
S_ACT.PGNO2=SDEFAULT.PGNO2
S_ACT.PRESS1=SDEFAULT.PRESS1
S_ACT.PRESS2=SDEFAULT.PRESS2
S_READY=FALSE
LIN XSWP_60_8398
USERSPOT(#SPOT, S_ACT)
WAIT FOR S_READY
;ENDFOLD

;FOLD ; SWP_60_8496;%{PE}%R 4.1.16,%MKUKATPBASIS,%CCOMMENT,%VNORMAL,%P 2:SWP_60_8496
;ENDFOLD
;FOLD LIN SWP_60_8496 L_OLP38 SPOT Gun=2 RETR OPN PgNo1=188 ACTIVE=1 NORMAL Tool[3]:Pinca C2 Base[3]:Atego/Axor;%{PE}%R 8.2.2,%MKUKATPSPOT,%CSPOT,%VLIN,%P 1:LIN, 2:SWP_60_8496, 3:, 5:2, 7:L_OLP38, 10:2, 12:#FIRST, 14:#OPN, 16:188, 18:1, 20:0, 22:0, 24:1, 25:NORMAL
$BWDSTART=FALSE
LDAT_ACT=LL_OLP38
FDAT_ACT=FSWP_60_8496
BAS(#CP_PARAMS,LL_OLP38.VEL)
S_ACT.GUN=2
S_ACT.PAIR=SDEFAULT.PAIR
S_ACT.RETR=#OPN
S_ACT.CLO_TM=1
S_ACT.PGNO1=188
S_ACT.PGNO2=SDEFAULT.PGNO2
S_ACT.PRESS1=SDEFAULT.PRESS1
S_ACT.PRESS2=SDEFAULT.PRESS2
S_READY=FALSE
LIN XSWP_60_8496
USERSPOT(#SPOT, S_ACT)
WAIT FOR S_READY
;ENDFOLD

;FOLD LIN l100 CONT Vel=2 m/s L_OLP39 Tool[3]:Pinca C2 Base[3]:Atego/Axor;%{PE}%R 8.2.20,%MKUKATPBASIS,%CMOVE,%VLIN,%P 1:LIN, 2:l100, 3:C_DIS C_DIS, 5:2, 7:L_OLP39
$BWDSTART=FALSE
LDAT_ACT=LL_OLP39
FDAT_ACT=Fl100
BAS(#CP_PARAMS,2)
LIN Xl100 C_DIS C_DIS
;ENDFOLD
;FOLD LIN l105 CONT Vel=2 m/s L_OLP40 Tool[3]:Pinca C2 Base[3]:Atego/Axor;%{PE}%R 8.2.20,%MKUKATPBASIS,%CMOVE,%VLIN,%P 1:LIN, 2:l105, 3:C_DIS C_DIS, 5:2, 7:L_OLP40
$BWDSTART=FALSE
LDAT_ACT=LL_OLP40
FDAT_ACT=Fl105
BAS(#CP_PARAMS,2)
LIN Xl105 C_DIS C_DIS
;ENDFOLD
;FOLD PTP l110 CONT Vel=100 % PDAT1 Tool[3]:Pinca C2 Base[3]:Atego/Axor;%{PE}%R 8.2.20,%MKUKATPBASIS,%CMOVE,%VPTP,%P 1:PTP, 2:l110, 3:C_DIS, 5:100, 7:PDAT1
$BWDSTART=FALSE
PDAT_ACT=PPDAT1
FDAT_ACT=Fl110
BAS(#PTP_PARAMS,100)
PTP Xl110 C_DIS
;ENDFOLD
;FOLD PTP l115 Vel=100 % P_OLP2 Tool[3]:Pinca C2 Base[3]:Atego/Axor;%{PE}%R 8.2.20,%MKUKATPBASIS,%CMOVE,%VPTP,%P 1:PTP, 2:l115, 3:, 5:100, 7:P_OLP2
$BWDSTART=FALSE
PDAT_ACT=PP_OLP2
FDAT_ACT=Fl115
BAS(#PTP_PARAMS,100)
PTP Xl115
;ENDFOLD

IF (NOT(GHOST())) THEN
IF FraesAnf(3) THEN
f_Fraes3 ()
ENDIF
ENDIF

END

--- ps_b_ltb_res_c02.dat ---
&ACCESS RVO1
&COMMENT Solda Axor LTB
&PARAM DISKPATH = KRC:\R1\Program\OLP
DEFDAT ps_b_ltb_res_c02
;FOLD EXTERNAL DECLARATIONS;%{PE}%MKUKATPBASIS,%CEXT,%VCOMMON,%P
;FOLD GRIPPERTECH EXT
EXT  H50 (INT  :IN,INT  :IN,INT  :IN,GRP_TYP  :IN )
;ENDFOLD (GRIPPERTECH EXT)
;FOLD SPOTTECH EXT
EXT  USERSPOT (S_COMMAND  :IN,SPOT_TYPE  :IN )
;ENDFOLD (SPOTTECH EXT)
;FOLD BASISTECH EXT;%{PE}%MKUKATPBASIS,%CEXT,%VEXT,%P
EXT  BAS (BAS_COMMAND  :IN,REAL  :IN )
DECL INT SUCCESS
;ENDFOLD (BASISTECH EXT)
;FOLD USER EXT;%{E}%MKUKATPUSER,%CEXT,%VEXT,%P
;Make your modifications here

;ENDFOLD (USER EXT)
;ENDFOLD (EXTERNAL DECLARATIONS)
DECL FDAT Fl010={TOOL_NO 3,BASE_NO 3,IPO_FRAME #BASE,POINT2[] " "}
DECL E6POS Xl010={X 137.790894,Y 755.423828,Z 801.72998,A 158.771606,B 69.1498032,C 162.299606,S 18,T 42,E1 0.0,E2 0.0,E3 0.0,E4 0.0,E5 0.0,E6 0.0}
DECL LDAT LL_OLP2={VEL 2.0,ACC 100.0,APO_DIST 10.0,APO_FAC 0.0,ORI_TYP #VAR,CIRC_TYP #BASE,JERK_FAC 50.0}
DECL FDAT Fl015={TOOL_NO 3,BASE_NO 3,IPO_FRAME #BASE,POINT2[] " "}
DECL E6POS Xl015={X 603.140991,Y 808.36499,Z 1241.97498,A 158.485001,B 12.9363003,C 166.735794,S 2,T 42}
DECL LDAT LL_OLP3={VEL 2.0,ACC 100.0,APO_DIST 10.0,APO_FAC 0.0,ORI_TYP #VAR,CIRC_TYP #BASE,JERK_FAC 50.0}
DECL FDAT Fl020={TOOL_NO 3,BASE_NO 3,IPO_FRAME #BASE,POINT2[] " "}
DECL E6POS Xl020={X 583.611084,Y 712.594788,Z 1181.354,A 154.968796,B 9.37294292,C 157.367905,S 18,T 42,E1 0.0,E2 0.0,E3 0.0,E4 0.0,E5 0.0,E6 0.0}
DECL LDAT LL_OLP4={VEL 2.0,ACC 100.0,APO_DIST 10.0,APO_FAC 0.0,ORI_TYP #VAR,CIRC_TYP #BASE,JERK_FAC 50.0}
DECL FDAT Fl025={TOOL_NO 3,BASE_NO 3,IPO_FRAME #BASE,POINT2[] " "}
DECL E6POS Xl025={X 570.496277,Y 697.463013,Z 1145.79199,A 154.968597,B 9.37284756,C 147.3685,S 18,T 42,E1 0.0,E2 0.0,E3 0.0,E4 0.0,E5 0.0,E6 0.0}
DECL LDAT LL_OLP5={VEL 2.0,ACC 100.0,APO_DIST 10.0,APO_FAC 0.0,ORI_TYP #VAR,CIRC_TYP #BASE,JERK_FAC 50.0}
DECL FDAT Fl030={TOOL_NO 3,BASE_NO 3,IPO_FRAME #BASE,POINT2[] " "}
DECL E6POS Xl030={X 582.752014,Y 1585.71301,Z 1144.11096,A 154.969406,B 9.37310028,C 157.3685,S 2,T 42}
DECL LDAT LL_OLP6={VEL 2.0,ACC 100.0,APO_DIST 10.0,APO_FAC 0.0,ORI_TYP #VAR,CIRC_TYP #BASE,JERK_FAC 50.0}
DECL FDAT Fl035={TOOL_NO 3,BASE_NO 3,IPO_FRAME #BASE,POINT2[] " "}
DECL E6POS Xl035={X 897.794006,Y 1320.91504,Z 1221.96802,A -149.936798,B -80.7937012,C 61.0237007,S 2,T 34}
DECL LDAT LL_OLP7={VEL 2.0,ACC 100.0,APO_DIST 30.0,APO_FAC 0.0,ORI_TYP #VAR,CIRC_TYP #BASE,JERK_FAC 50.0}
DECL FDAT Fl040={TOOL_NO 3,BASE_NO 3,IPO_FRAME #BASE,POINT2[] " "}
DECL E6POS Xl040={X 637.291992,Y 987.916992,Z 1221.96594,A -149.936798,B -80.7937012,C 61.0236015,S 2,T 34}
DECL LDAT LL_OLP8={VEL 2.0,ACC 100.0,APO_DIST 2.0,APO_FAC 0.0,ORI_TYP #VAR,CIRC_TYP #BASE,JERK_FAC 50.0}
DECL FDAT Fl045={TOOL_NO 3,BASE_NO 3,IPO_FRAME #BASE,POINT2[] " "}
DECL E6POS Xl045={X 597.394775,Y 971.886719,Z 1312.26404,A -116.101997,B -85.0568771,C 22.43223,S 18,T 34,E1 0.0,E2 0.0,E3 0.0,E4 0.0,E5 0.0,E6 0.0}
DECL LDAT LL_OLP9={VEL 2.0,ACC 100.0,APO_DIST 0.0,APO_FAC 0.0,ORI_TYP #VAR,CIRC_TYP #BASE,JERK_FAC 50.0}
DECL FDAT FSWP_60_8580={TOOL_NO 3,BASE_NO 3,IPO_FRAME #BASE,POINT2[] " "}
DECL E6POS XSWP_60_8580={X 594.508423,Y 984.949219,Z 1318.19995,A -158.478806,B -86.9592972,C 65.262207,S 18,T 34,E1 0.0,E2 0.0,E3 0.0,E4 0.0,E5 0.0,E6 0.0}
DECL LDAT LL_OLP10={VEL 2.0,ACC 100.0,APO_DIST 0.0,APO_FAC 0.0,ORI_TYP #VAR,CIRC_TYP #BASE,JERK_FAC 50.0}
DECL FDAT FSWP_60_8578={TOOL_NO 3,BASE_NO 3,IPO_FRAME #BASE,POINT2[] " "}
DECL E6POS XSWP_60_8578={X 622.711914,Y 985.182617,Z 1319.24695,A 140.782898,B -87.3470688,C 128.908401,S 18,T 34,E1 0.0,E2 0.0,E3 0.0,E4 0.0,E5 0.0,E6 0.0}
DECL LDAT LL_OLP11={VEL 2.0,ACC 100.0,APO_DIST 0.0,APO_FAC 0.0,ORI_TYP #VAR,CIRC_TYP #BASE,JERK_FAC 50.0}
DECL FDAT FSWP_60_8590={TOOL_NO 3,BASE_NO 3,IPO_FRAME #BASE,POINT2[] " "}
DECL E6POS XSWP_60_8590={X 649.788879,Y 983.73468,Z 1320.13403,A 149.639008,B -87.5716095,C 121.578499,S 18,T 34,E1 0.0,E2 0.0,E3 0.0,E4 0.0,E5 0.0,E6 0.0}
DECL LDAT LL_OLP12={VEL 2.0,ACC 100.0,APO_DIST 0.0,APO_FAC 0.0,ORI_TYP #VAR,CIRC_TYP #BASE,JERK_FAC 50.0}
DECL FDAT Fl050={TOOL_NO 3,BASE_NO 3,IPO_FRAME #BASE,POINT2[] " "}
DECL E6POS Xl050={X 660.460388,Y 983.00177,Z 1317.37402,A -113.609398,B -85.0964127,C 24.9298801,S 18,T 34,E1 0.0,E2 0.0,E3 0.0,E4 0.0,E5 0.0,E6 0.0}
DECL LDAT LL_OLP13={VEL 2.0,ACC 100.0,APO_DIST 2.0,APO_FAC 0.0,ORI_TYP #VAR,CIRC_TYP #BASE,JERK_FAC 50.0}
DECL FDAT Fl060={TOOL_NO 3,BASE_NO 3,IPO_FRAME #BASE,POINT2[] " "}
DECL E6POS Xl060={X 1323.12305,Y 1352.31897,Z 35.6313095,A -179.994003,B -18.8152809,C 89.9956131,S 18,T 34,E1 0.0,E2 0.0,E3 0.0,E4 0.0,E5 0.0,E6 0.0}
DECL LDAT LL_OLP15={VEL 2.0,ACC 100.0,APO_DIST 30.0,APO_FAC 0.0,ORI_TYP #VAR,CIRC_TYP #BASE,JERK_FAC 50.0}
DECL FDAT Fl075={TOOL_NO 3,BASE_NO 3,IPO_FRAME #BASE,POINT2[] " "}
DECL E6POS Xl075={X 1319.21802,Y 1023.45697,Z 114.155502,A 179.976303,B -22.25774,C 89.9964523,S 18,T 34,E1 0.0,E2 0.0,E3 0.0,E4 0.0,E5 0.0,E6 0.0}
DECL LDAT LL_OLP18={VEL 2.0,ACC 100.0,APO_DIST 0.0,APO_FAC 0.0,ORI_TYP #VAR,CIRC_TYP #BASE,JERK_FAC 50.0}
DECL FDAT FSWP_60_8532={TOOL_NO 3,BASE_NO 3,IPO_FRAME #BASE,POINT2[] " "}
DECL E6POS XSWP_60_8532={X 1316.25903,Y 1033.04004,Z 113.953598,A 179.772095,B -22.2714405,C 89.0541229,S 18,T 34,E1 0.0,E2 0.0,E3 0.0,E4 0.0,E5 0.0,E6 0.0}
DECL LDAT LL_OLP19={VEL 2.0,ACC 100.0,APO_DIST 0.0,APO_FAC 0.0,ORI_TYP #VAR,CIRC_TYP #BASE,JERK_FAC 50.0}
DECL FDAT FSWP_60_8530={TOOL_NO 3,BASE_NO 3,IPO_FRAME #BASE,POINT2[] " "}
DECL E6POS XSWP_60_8530={X 1360.77295,Y 1030.79602,Z 114.927902,A 179.979202,B -22.3133202,C 90.9138718,S 18,T 34,E1 0.0,E2 0.0,E3 0.0,E4 0.0,E5 0.0,E6 0.0}
DECL LDAT LL_OLP20={VEL 2.0,ACC 100.0,APO_DIST 0.0,APO_FAC 0.0,ORI_TYP #VAR,CIRC_TYP #BASE,JERK_FAC 50.0}
DECL FDAT FSWP_60_8528={TOOL_NO 3,BASE_NO 3,IPO_FRAME #BASE,POINT2[] " "}
DECL E6POS XSWP_60_8528={X 1401.98096,Y 1031.41699,Z 115.391502,A 179.656601,B -22.3331699,C 91.4622269,S 18,T 34,E1 0.0,E2 0.0,E3 0.0,E4 0.0,E5 0.0,E6 0.0}
DECL LDAT LL_OLP21={VEL 2.0,ACC 100.0,APO_DIST 0.0,APO_FAC 0.0,ORI_TYP #VAR,CIRC_TYP #BASE,JERK_FAC 50.0}
DECL FDAT Fl080={TOOL_NO 3,BASE_NO 3,IPO_FRAME #BASE,POINT2[] " "}
DECL E6POS Xl080={X 1417.18701,Y 1021.49597,Z 96.9904327,A 179.976395,B -22.3135891,C 89.9944611,S 18,T 34,E1 0.0,E2 0.0,E3 0.0,E4 0.0,E5 0.0,E6 0.0}
DECL LDAT LL_OLP22={VEL 2.0,ACC 100.0,APO_DIST 3.0,APO_FAC 0.0,ORI_TYP #VAR,CIRC_TYP #BASE,JERK_FAC 50.0}
DECL FDAT Fl085={TOOL_NO 3,BASE_NO 3,IPO_FRAME #BASE,POINT2[] " "}
DECL E6POS Xl085={X 1478.59302,Y 1018.30701,Z 107.972801,A 179.981995,B -21.8126202,C 91.8198471,S 18,T 34,E1 0.0,E2 0.0,E3 0.0,E4 0.0,E5 0.0,E6 0.0}
DECL LDAT LL_OLP23={VEL 2.0,ACC 100.0,APO_DIST 3.0,APO_FAC 0.0,ORI_TYP #VAR,CIRC_TYP #BASE,JERK_FAC 50.0}
DECL FDAT FSWP_60_8524={TOOL_NO 3,BASE_NO 3,IPO_FRAME #BASE,POINT2[] " "}
DECL E6POS XSWP_60_8524={X 1481.91003,Y 1027.86096,Z 116.624199,A 179.983902,B -21.8115196,C 94.6476288,S 18,T 42,E1 0.0,E2 0.0,E3 0.0,E4 0.0,E5 0.0,E6 0.0}
DECL LDAT LL_OLP24={VEL 2.0,ACC 100.0,APO_DIST 0.0,APO_FAC 0.0,ORI_TYP #VAR,CIRC_TYP #BASE,JERK_FAC 50.0}
DECL FDAT FSWP_60_8522={TOOL_NO 3,BASE_NO 3,IPO_FRAME #BASE,POINT2[] " "}
DECL E6POS XSWP_60_8522={X 1519.79395,Y 1027.22595,Z 116.093903,A 179.9823,B -21.8113403,C 94.0460892,S 18,T 42,E1 0.0,E2 0.0,E3 0.0,E4 0.0,E5 0.0,E6 0.0}
DECL LDAT LL_OLP25={VEL 2.0,ACC 100.0,APO_DIST 0.0,APO_FAC 0.0,ORI_TYP #VAR,CIRC_TYP #BASE,JERK_FAC 50.0}
DECL FDAT FSWP_60_8520={TOOL_NO 3,BASE_NO 3,IPO_FRAME #BASE,POINT2[] " "}
DECL E6POS XSWP_60_8520={X 1559.94702,Y 1025.41394,Z 114.939697,A 179.989197,B -21.8192997,C 93.8743362,S 18,T 42,E1 0.0,E2 0.0,E3 0.0,E4 0.0,E5 0.0,E6 0.0}
DECL LDAT LL_OLP26={VEL 2.0,ACC 100.0,APO_DIST 0.0,APO_FAC 0.0,ORI_TYP #VAR,CIRC_TYP #BASE,JERK_FAC 50.0}
DECL FDAT FSWP_60_8516={TOOL_NO 3,BASE_NO 3,IPO_FRAME #BASE,POINT2[] " "}
DECL E6POS XSWP_60_8516={X 1623.01404,Y 1024.82397,Z 114.182503,A 179.982101,B -21.8135796,C 93.8866425,S 18,T 42,E1 0.0,E2 0.0,E3 0.0,E4 0.0,E5 0.0,E6 0.0}
DECL LDAT LL_OLP29={VEL 2.0,ACC 100.0,APO_DIST 0.0,APO_FAC 0.0,ORI_TYP #VAR,CIRC_TYP #BASE,JERK_FAC 50.0}
DECL FDAT FSWP_60_8514={TOOL_NO 3,BASE_NO 3,IPO_FRAME #BASE,POINT2[] " "}
DECL E6POS XSWP_60_8514={X 1665.75195,Y 1025.18201,Z 114.200699,A 179.981995,B -21.8153095,C 94.3753433,S 18,T 42,E1 0.0,E2 0.0,E3 0.0,E4 0.0,E5 0.0,E6 0.0}
DECL LDAT LL_OLP30={VEL 2.0,ACC 100.0,APO_DIST 0.0,APO_FAC 0.0,ORI_TYP #VAR,CIRC_TYP #BASE,JERK_FAC 50.0}
DECL FDAT FSWP_60_8512={TOOL_NO 3,BASE_NO 3,IPO_FRAME #BASE,POINT2[] " "}
DECL E6POS XSWP_60_8512={X 1712.14697,Y 1024.44995,Z 112.631699,A 179.985107,B -21.8173199,C 94.0283585,S 18,T 34,E1 0.0,E2 0.0,E3 0.0,E4 0.0,E5 0.0,E6 0.0}
DECL LDAT LL_OLP31={VEL 2.0,ACC 100.0,APO_DIST 0.0,APO_FAC 0.0,ORI_TYP #VAR,CIRC_TYP #BASE,JERK_FAC 50.0}
DECL FDAT FSWP_60_8510={TOOL_NO 3,BASE_NO 3,IPO_FRAME #BASE,POINT2[] " "}
DECL E6POS XSWP_60_8510={X 1759.86304,Y 1023.995,Z 110.8787,A 179.981293,B -21.8202209,C 93.9407806,S 18,T 34,E1 0.0,E2 0.0,E3 0.0,E4 0.0,E5 0.0,E6 0.0}
DECL LDAT LL_OLP32={VEL 2.0,ACC 100.0,APO_DIST 0.0,APO_FAC 0.0,ORI_TYP #VAR,CIRC_TYP #BASE,JERK_FAC 50.0}
DECL FDAT FSWP_60_8508={TOOL_NO 3,BASE_NO 3,IPO_FRAME #BASE,POINT2[] " "}
DECL E6POS XSWP_60_8508={X 1809.09705,Y 1023.68903,Z 108.639397,A 179.981201,B -21.8179302,C 94.7481766,S 18,T 42,E1 0.0,E2 0.0,E3 0.0,E4 0.0,E5 0.0,E6 0.0}
DECL LDAT LL_OLP33={VEL 2.0,ACC 100.0,APO_DIST 0.0,APO_FAC 0.0,ORI_TYP #VAR,CIRC_TYP #BASE,JERK_FAC 50.0}
DECL FDAT FSWP_60_8504={TOOL_NO 3,BASE_NO 3,IPO_FRAME #BASE,POINT2[] " "}
DECL E6POS XSWP_60_8504={X 1909.02502,Y 1021.68903,Z 105.446701,A 179.983704,B -21.8215504,C 90.8531494,S 18,T 34,E1 0.0,E2 0.0,E3 0.0,E4 0.0,E5 0.0,E6 0.0}
DECL LDAT LL_OLP34={VEL 2.0,ACC 100.0,APO_DIST 0.0,APO_FAC 0.0,ORI_TYP #VAR,CIRC_TYP #BASE,JERK_FAC 50.0}
DECL FDAT FSWP_60_8502={TOOL_NO 3,BASE_NO 3,IPO_FRAME #BASE,POINT2[] " "}
DECL E6POS XSWP_60_8502={X 1961.62903,Y 1019.48401,Z 104.019402,A 179.9785,B -21.8217201,C 91.1027832,S 18,T 34,E1 0.0,E2 0.0,E3 0.0,E4 0.0,E5 0.0,E6 0.0}
DECL LDAT LL_OLP35={VEL 2.0,ACC 100.0,APO_DIST 0.0,APO_FAC 0.0,ORI_TYP #VAR,CIRC_TYP #BASE,JERK_FAC 50.0}
DECL FDAT FSWP_60_8500={TOOL_NO 3,BASE_NO 3,IPO_FRAME #BASE,POINT2[] " "}
DECL E6POS XSWP_60_8500={X 2024.10596,Y 1020.47498,Z 101.323097,A -179.814697,B -21.6788292,C 93.8341064,S 18,T 34,E1 0.0,E2 0.0,E3 0.0,E4 0.0,E5 0.0,E6 0.0}
DECL LDAT LL_OLP36={VEL 2.0,ACC 100.0,APO_DIST 0.0,APO_FAC 0.0,ORI_TYP #VAR,CIRC_TYP #BASE,JERK_FAC 50.0}
DECL FDAT FSWP_60_8498={TOOL_NO 3,BASE_NO 3,IPO_FRAME #BASE,POINT2[] " "}
DECL E6POS XSWP_60_8498={X 2087.2439,Y 1019.17603,Z 101.204903,A 179.832703,B -24.38311,C 92.6964569,S 18,T 34,E1 0.0,E2 0.0,E3 0.0,E4 0.0,E5 0.0,E6 0.0}
DECL LDAT LL_OLP37={VEL 2.0,ACC 100.0,APO_DIST 0.0,APO_FAC 0.0,ORI_TYP #VAR,CIRC_TYP #BASE,JERK_FAC 50.0}
DECL FDAT FSWP_60_8496={TOOL_NO 3,BASE_NO 3,IPO_FRAME #BASE,POINT2[] " "}
DECL E6POS XSWP_60_8496={X 2153.47705,Y 1017.854,Z 101.577003,A 179.2276,B -38.2940292,C 92.0559082,S 18,T 34,E1 0.0,E2 0.0,E3 0.0,E4 0.0,E5 0.0,E6 0.0}
DECL LDAT LL_OLP38={VEL 2.0,ACC 100.0,APO_DIST 0.0,APO_FAC 0.0,ORI_TYP #VAR,CIRC_TYP #BASE,JERK_FAC 50.0}
DECL FDAT Fl100={TOOL_NO 3,BASE_NO 3,IPO_FRAME #BASE,POINT2[] " "}
DECL E6POS Xl100={X 2124.13599,Y 1014.198,Z 40.5825882,A 179.976501,B -21.8289909,C 91.8177567,S 18,T 34,E1 0.0,E2 0.0,E3 0.0,E4 0.0,E5 0.0,E6 0.0}
DECL LDAT LL_OLP39={VEL 2.0,ACC 100.0,APO_DIST 5.0,APO_FAC 0.0,ORI_TYP #VAR,CIRC_TYP #BASE,JERK_FAC 50.0}
DECL FDAT Fl105={TOOL_NO 3,BASE_NO 3,IPO_FRAME #BASE,POINT2[] " "}
DECL E6POS Xl105={X 1973.10205,Y 1113.71301,Z 22.7551403,A -177.173203,B -26.8758907,C 89.4126968,S 18,T 34,E1 0.0,E2 0.0,E3 0.0,E4 0.0,E5 0.0,E6 0.0}
DECL LDAT LL_OLP40={VEL 2.0,ACC 100.0,APO_DIST 30.0,APO_FAC 0.0,ORI_TYP #VAR,CIRC_TYP #BASE,JERK_FAC 50.0}
DECL FDAT Fl110={TOOL_NO 3,BASE_NO 3,IPO_FRAME #BASE,POINT2[] " "}
DECL E6POS Xl110={X 1765.68298,Y 1252.62695,Z 49.1746597,A -178.002701,B -30.1959591,C 89.5175018,S 18,T 34,E1 0.0,E2 0.0,E3 0.0,E4 0.0,E5 0.0,E6 0.0}
DECL FDAT Fl115={TOOL_NO 3,BASE_NO 3,IPO_FRAME #BASE,POINT2[] " "}
DECL PDAT PP_OLP2={VEL 100.0,ACC 100.0,APO_DIST 100.0,APO_MODE #CDIS}
DECL E6POS Xl115={X 1738.02795,Y 2276.4519,Z 99.2014771,A 178.272095,B -17.5484295,C 90.5386963,S 18,T 42,E1 0.0,E2 0.0,E3 0.0,E4 0.0,E5 0.0,E6 0.0}
DECL BASIS_SUGG_T LAST_BASIS={POINT1[] "P0                      ",POINT2[] "P0                      ",CP_PARAMS[] "CPDAT0                  ",PTP_PARAMS[] "PDAT0                   ",CONT[] "                        ",CP_VEL[] "2.0                     ",PTP_VEL[] " 100                    ",SYNC_PARAMS[] "SYNCDAT                 ",SPL_NAME[] "S0                      "}
DECL E6POS XSWP_60_8790={X 723.895081,Y 983.757813,Z 1322.13794,A 8.92934895,B -75.0166016,C -96.2660828,S 18,T 34,E1 0.0,E2 0.0,E3 0.0,E4 0.0,E5 0.0,E6 0.0}

DECL FDAT FSWP_60_8790={TOOL_NO 3,BASE_NO 3,IPO_FRAME #BASE,POINT2[] " "}

DECL E6POS XSWP_60_8792={X 760.629028,Y 985.101013,Z 1322.11401,A 4.67850685,B -75.0971069,C -92.1634827,S 18,T 34,E1 0.0,E2 0.0,E3 0.0,E4 0.0,E5 0.0,E6 0.0}

DECL FDAT FSWP_60_8792={TOOL_NO 3,BASE_NO 3,IPO_FRAME #BASE,POINT2[] " "}

DECL E6POS XSWP_60_8794={X 800.937927,Y 985.885193,Z 1321.32605,A 4.28598499,B -75.2968826,C -91.2004471,S 18,T 34,E1 0.0,E2 0.0,E3 0.0,E4 0.0,E5 0.0,E6 0.0}

DECL FDAT FSWP_60_8794={TOOL_NO 3,BASE_NO 3,IPO_FRAME #BASE,POINT2[] " "}

DECL E6POS XSWP_60_8796={X 847.146912,Y 986.669678,Z 1322.81201,A -7.07662487,B -75.2146225,C -79.7810898,S 18,T 34,E1 0.0,E2 0.0,E3 0.0,E4 0.0,E5 0.0,E6 0.0}

DECL FDAT FSWP_60_8796={TOOL_NO 3,BASE_NO 3,IPO_FRAME #BASE,POINT2[] " "}


DECL E6POS XSWP_60_8798={X 903.060974,Y 987.891174,Z 1322.86096,A -5.14305401,B -75.1807632,C -81.9936905,S 18,T 34,E1 0.0,E2 0.0,E3 0.0,E4 0.0,E5 0.0,E6 0.0}
DECL FDAT FSWP_60_8798={TOOL_NO 3,BASE_NO 3,IPO_FRAME #BASE,POINT2[] " "}

DECL E6POS XSWP_60_8802={X 1004.84601,Y 986.23053,Z 1321.85303,A -9.05966473,B -74.9902267,C -78.2642136,S 18,T 34,E1 0.0,E2 0.0,E3 0.0,E4 0.0,E5 0.0,E6 0.0}

DECL FDAT FSWP_60_8802={TOOL_NO 3,BASE_NO 3,IPO_FRAME #BASE,POINT2[] " "}

DECL E6POS XSWP_60_8804={X 1056.08704,Y 987.01947,Z 1321.62,A -9.69501877,B -74.9384079,C -77.704628,S 18,T 34,E1 0.0,E2 0.0,E3 0.0,E4 0.0,E5 0.0,E6 0.0}

DECL FDAT FSWP_60_8804={TOOL_NO 3,BASE_NO 3,IPO_FRAME #BASE,POINT2[] " "}


DECL E6POS XSWP_60_8806={X 1105.448,Y 986.423279,Z 1321.96997,A -11.5182104,B -74.7811737,C -76.1092072,S 18,T 34,E1 0.0,E2 0.0,E3 0.0,E4 0.0,E5 0.0,E6 0.0}
DECL FDAT FSWP_60_8806={TOOL_NO 3,BASE_NO 3,IPO_FRAME #BASE,POINT2[] " "}
DECL E6POS XSWP_60_8808={X 1143.96399,Y 986.294922,Z 1320.552,A -9.89994812,B -74.9099808,C -77.5606003,S 18,T 34,E1 0.0,E2 0.0,E3 0.0,E4 0.0,E5 0.0,E6 0.0}
DECL FDAT FSWP_60_8808={TOOL_NO 3,BASE_NO 3,IPO_FRAME #BASE,POINT2[] " "}

DECL E6POS XSWP_60_8810={X 1183.86401,Y 986.277588,Z 1319.65796,A -3.22921395,B -75.0366821,C -84.5194931,S 18,T 34,E1 0.0,E2 0.0,E3 0.0,E4 0.0,E5 0.0,E6 0.0}
DECL FDAT FSWP_60_8810={TOOL_NO 3,BASE_NO 3,IPO_FRAME #BASE,POINT2[] " "}
DECL PDAT PP_OLP4={VEL 100.0,ACC 100.0,APO_DIST 30.0,APO_MODE #CDIS}
DECL E6POS Xl006={X 1083.797,Y 1451.30701,Z 836.236023,A 174.173294,B -30.1965008,C 118.184799,S 2,T 42}
DECL FDAT Fl006={TOOL_NO 3,BASE_NO 3,IPO_FRAME #BASE,POINT2[] " "}
DECL LDAT LL_OLP48={VEL 2.0,ACC 100.0,APO_DIST 30.0,APO_FAC 0.0,ORI_TYP #VAR,CIRC_TYP #BASE,JERK_FAC 50.0}
DECL E6POS Xl011={X 563.752014,Y 1566.71301,Z 1132.11096,A 154.969406,B 9.37310028,C 157.3685,S 2,T 42}
DECL FDAT Fl011={TOOL_NO 3,BASE_NO 3,IPO_FRAME #BASE,POINT2[] " "}
DECL LDAT LL_OLP49={VEL 2.0,ACC 100.0,APO_DIST 10.0,APO_FAC 0.0,ORI_TYP #VAR,CIRC_TYP #BASE,JERK_FAC 50.0}
DECL E6POS Xl016={X 562.511414,Y 691.50061,Z 1119.09802,A 154.969101,B 9.37301254,C 147.368195,S 18,T 42,E1 0.0,E2 0.0,E3 0.0,E4 0.0,E5 0.0,E6 0.0}
DECL FDAT Fl016={TOOL_NO 3,BASE_NO 3,IPO_FRAME #BASE,POINT2[] " "}
DECL PDAT PP_OLP5={VEL 100.0,ACC 100.0,APO_DIST 10.0,APO_MODE #CDIS}
DECL E6POS Xl021={X 564.166016,Y 693.661499,Z 1150.06299,A 154.969101,B 9.37302113,C 157.368195,S 18,T 42,E1 0.0,E2 0.0,E3 0.0,E4 0.0,E5 0.0,E6 0.0}
DECL FDAT Fl021={TOOL_NO 3,BASE_NO 3,IPO_FRAME #BASE,POINT2[] " "}
DECL LDAT LL_OLP50={VEL 2.0,ACC 100.0,APO_DIST 10.0,APO_FAC 0.0,ORI_TYP #VAR,CIRC_TYP #BASE,JERK_FAC 50.0}
DECL E6POS Xl026={X 582.596375,Y 789.625122,Z 1163.21899,A 158.486099,B 12.9365396,C 166.737305,S 18,T 42,E1 0.0,E2 0.0,E3 0.0,E4 0.0,E5 0.0,E6 0.0}
DECL FDAT Fl026={TOOL_NO 3,BASE_NO 3,IPO_FRAME #BASE,POINT2[] " "}
DECL LDAT LCPDAT0={VEL 2.0,ACC 100.0,APO_DIST 100.0,APO_FAC 50.0,AXIS_VEL 100.0,AXIS_ACC 100.0,ORI_TYP #VAR,CIRC_TYP #BASE,JERK_FAC 50.0,GEAR_JERK 50.0,EXAX_IGN 0}
DECL E6POS XP0={X 567.326416,Y 409.623993,Z 1234.31702,A 158.465195,B 12.93505,C 166.748199,S 18,T 42,E1 0.0,E2 0.0,E3 0.0,E4 0.0,E5 0.0,E6 0.0}
DECL FDAT FP0={TOOL_NO 3,BASE_NO 3,IPO_FRAME #BASE,POINT2[] " ",TQ_STATE FALSE}
DECL LDAT LCPDAT1={VEL 2.0,ACC 100.0,APO_DIST 100.0,APO_FAC 50.0,AXIS_VEL 100.0,AXIS_ACC 100.0,ORI_TYP #VAR,CIRC_TYP #BASE,JERK_FAC 50.0,GEAR_JERK 50.0,EXAX_IGN 0}
DECL E6POS XP1={X 622.916321,Y 355.254211,Z 1422.57605,A 157.948105,B 12.9317598,C 166.758606,S 18,T 42,E1 0.0,E2 0.0,E3 0.0,E4 0.0,E5 0.0,E6 0.0}
DECL FDAT FP1={TOOL_NO 3,BASE_NO 3,IPO_FRAME #BASE,POINT2[] " ",TQ_STATE FALSE}
DECL LDAT LCPDAT2={VEL 2.0,ACC 100.0,APO_DIST 30.0,APO_FAC 50.0,AXIS_VEL 100.0,AXIS_ACC 100.0,ORI_TYP #VAR,CIRC_TYP #BASE,JERK_FAC 50.0,GEAR_JERK 50.0,EXAX_IGN 0}
DECL E6POS XP2={X 539.093994,Y 258.427307,Z 1367.42297,A 155.131699,B 22.3258801,C 163.030502,S 18,T 42,E1 0.0,E2 0.0,E3 0.0,E4 0.0,E5 0.0,E6 0.0}
DECL FDAT FP2={TOOL_NO 3,BASE_NO 3,IPO_FRAME #BASE,POINT2[] " ",TQ_STATE FALSE}
DECL LDAT LCPDAT3={VEL 2.0,ACC 100.0,APO_DIST 10.0,APO_FAC 50.0,AXIS_VEL 100.0,AXIS_ACC 100.0,ORI_TYP #VAR,CIRC_TYP #BASE,JERK_FAC 50.0,GEAR_JERK 50.0,EXAX_IGN 0}
DECL E6POS XP3={X 400.828705,Y 277.572998,Z 1191.0,A 150.367203,B 35.5739708,C 156.604507,S 18,T 42,E1 0.0,E2 0.0,E3 0.0,E4 0.0,E5 0.0,E6 0.0}
DECL FDAT FP3={TOOL_NO 3,BASE_NO 3,IPO_FRAME #BASE,POINT2[] " ",TQ_STATE FALSE}
DECL LDAT LL_OLP51={VEL 2.0,ACC 100.0,APO_DIST 10.0,APO_FAC 0.0,ORI_TYP #VAR,CIRC_TYP #BASE,JERK_FAC 50.0}
DECL E6POS Xl031={X 350.266815,Y 288.423492,Z 1120.07996,A 150.391205,B 43.1624107,C 155.955505,S 18,T 42,E1 0.0,E2 0.0,E3 0.0,E4 0.0,E5 0.0,E6 0.0}
DECL FDAT Fl031={TOOL_NO 3,BASE_NO 3,IPO_FRAME #BASE,POINT2[] " "}
DECL PDAT PP_OLP6={VEL 100.0,ACC 100.0,APO_DIST 0.0,APO_MODE #CDIS}
DECL E6POS Xl036={X 317.7453,Y 296.586395,Z 1050.84399,A 147.642303,B 47.8915787,C 153.828995,S 18,T 42,E1 0.0,E2 0.0,E3 0.0,E4 0.0,E5 0.0,E6 0.0}
DECL FDAT Fl036={TOOL_NO 3,BASE_NO 3,IPO_FRAME #BASE,POINT2[] " "}
DECL PDAT PP_OLP7={VEL 100.0,ACC 100.0,APO_DIST 5.0,APO_MODE #CDIS}
DECL E6POS Xl041={X 102.250198,Y 340.10611,Z 682.652588,A 164.808105,B 79.9921112,C 167.133606,S 18,T 42,E1 0.0,E2 0.0,E3 0.0,E4 0.0,E5 0.0,E6 0.0}
DECL FDAT Fl041={TOOL_NO 3,BASE_NO 3,IPO_FRAME #BASE,POINT2[] " "}
DECL LDAT LL_OLP52={VEL 2.0,ACC 100.0,APO_DIST 5.0,APO_FAC 0.0,ORI_TYP #VAR,CIRC_TYP #BASE,JERK_FAC 50.0}
DECL E6POS Xl046={X 71.2702866,Y 356.045807,Z 624.529419,A 159.397202,B 82.8824234,C 161.778595,S 18,T 42,E1 0.0,E2 0.0,E3 0.0,E4 0.0,E5 0.0,E6 0.0}
DECL FDAT Fl046={TOOL_NO 3,BASE_NO 3,IPO_FRAME #BASE,POINT2[] " "}
DECL LDAT LL_OLP53={VEL 2.0,ACC 100.0,APO_DIST 0.0,APO_FAC 0.0,ORI_TYP #VAR,CIRC_TYP #BASE,JERK_FAC 50.0}
DECL E6POS XSWP_60_9280={X 93.7982178,Y 380.760986,Z 613.06543,A 159.360794,B 82.8838272,C 161.736404,S 18,T 42,E1 0.0,E2 0.0,E3 0.0,E4 0.0,E5 0.0,E6 0.0}
DECL FDAT FSWP_60_9280={TOOL_NO 3,BASE_NO 3,IPO_FRAME #BASE,POINT2[] " "}
DECL LDAT LL_OLP54={VEL 2.0,ACC 100.0,APO_DIST 0.0,APO_FAC 0.0,ORI_TYP #VAR,CIRC_TYP #BASE,JERK_FAC 50.0}
DECL E6POS XSWP_60_9282={X 95.1983414,Y 412.033203,Z 612.224121,A 159.370499,B 82.8822937,C 161.745895,S 18,T 42,E1 0.0,E2 0.0,E3 0.0,E4 0.0,E5 0.0,E6 0.0}
DECL FDAT FSWP_60_9282={TOOL_NO 3,BASE_NO 3,IPO_FRAME #BASE,POINT2[] " "}
DECL LDAT LL_OLP55={VEL 2.0,ACC 100.0,APO_DIST 0.0,APO_FAC 0.0,ORI_TYP #VAR,CIRC_TYP #BASE,JERK_FAC 50.0}
DECL E6POS XSWP_60_9286={X 98.8377228,Y 478.136993,Z 615.090515,A 158.5354,B 82.6687012,C 159.334305,S 18,T 42,E1 0.0,E2 0.0,E3 0.0,E4 0.0,E5 0.0,E6 0.0}
DECL FDAT FSWP_60_9286={TOOL_NO 3,BASE_NO 3,IPO_FRAME #BASE,POINT2[] " "}
DECL LDAT LL_OLP56={VEL 2.0,ACC 100.0,APO_DIST 0.0,APO_FAC 0.0,ORI_TYP #VAR,CIRC_TYP #BASE,JERK_FAC 50.0}
DECL E6POS XSWP_60_9288={X 100.442497,Y 513.4646,Z 616.12793,A 159.082596,B 82.9018936,C 159.794601,S 18,T 42,E1 0.0,E2 0.0,E3 0.0,E4 0.0,E5 0.0,E6 0.0}
DECL FDAT FSWP_60_9288={TOOL_NO 3,BASE_NO 3,IPO_FRAME #BASE,POINT2[] " "}
DECL LDAT LL_OLP57={VEL 2.0,ACC 100.0,APO_DIST 0.0,APO_FAC 0.0,ORI_TYP #VAR,CIRC_TYP #BASE,JERK_FAC 50.0}
DECL E6POS XSWP_60_9290={X 102.522003,Y 545.988403,Z 614.039917,A 160.234299,B 82.879837,C 161.132095,S 18,T 42,E1 0.0,E2 0.0,E3 0.0,E4 0.0,E5 0.0,E6 0.0}
DECL FDAT FSWP_60_9290={TOOL_NO 3,BASE_NO 3,IPO_FRAME #BASE,POINT2[] " "}
DECL LDAT LL_OLP58={VEL 2.0,ACC 100.0,APO_DIST 0.0,APO_FAC 0.0,ORI_TYP #VAR,CIRC_TYP #BASE,JERK_FAC 50.0}
DECL E6POS XSWP_60_9292={X 103.919098,Y 574.488892,Z 615.100891,A 159.7061,B 82.8799286,C 161.684998,S 18,T 42,E1 0.0,E2 0.0,E3 0.0,E4 0.0,E5 0.0,E6 0.0}
DECL FDAT FSWP_60_9292={TOOL_NO 3,BASE_NO 3,IPO_FRAME #BASE,POINT2[] " "}
DECL LDAT LL_OLP59={VEL 2.0,ACC 100.0,APO_DIST 0.0,APO_FAC 0.0,ORI_TYP #VAR,CIRC_TYP #BASE,JERK_FAC 50.0}
DECL E6POS XSWP_60_9296={X 108.416,Y 646.456177,Z 614.435181,A 159.410507,B 82.8830185,C 161.785904,S 18,T 42,E1 0.0,E2 0.0,E3 0.0,E4 0.0,E5 0.0,E6 0.0}
DECL FDAT FSWP_60_9296={TOOL_NO 3,BASE_NO 3,IPO_FRAME #BASE,POINT2[] " "}
DECL LDAT LL_OLP77={VEL 2.0,ACC 100.0,APO_DIST 0.0,APO_FAC 0.0,ORI_TYP #VAR,CIRC_TYP #BASE,JERK_FAC 50.0}
DECL E6POS XSWP_60_9298={X 111.716202,Y 682.766418,Z 615.322815,A 159.398407,B 82.8831482,C 161.775604,S 18,T 42,E1 0.0,E2 0.0,E3 0.0,E4 0.0,E5 0.0,E6 0.0}
DECL FDAT FSWP_60_9298={TOOL_NO 3,BASE_NO 3,IPO_FRAME #BASE,POINT2[] " "}
DECL LDAT LL_OLP78={VEL 2.0,ACC 100.0,APO_DIST 0.0,APO_FAC 0.0,ORI_TYP #VAR,CIRC_TYP #BASE,JERK_FAC 50.0}
DECL E6POS XSWP_60_9300={X 114.766197,Y 718.722412,Z 616.54657,A 159.434402,B 82.8802872,C 161.813995,S 18,T 42,E1 0.0,E2 0.0,E3 0.0,E4 0.0,E5 0.0,E6 0.0}
DECL FDAT FSWP_60_9300={TOOL_NO 3,BASE_NO 3,IPO_FRAME #BASE,POINT2[] " "}
DECL LDAT LL_OLP79={VEL 2.0,ACC 100.0,APO_DIST 0.0,APO_FAC 0.0,ORI_TYP #VAR,CIRC_TYP #BASE,JERK_FAC 50.0}
DECL E6POS XSWP_60_9302={X 119.6847,Y 754.768677,Z 617.763794,A 159.414795,B 82.8860092,C 161.790604,S 18,T 42,E1 0.0,E2 0.0,E3 0.0,E4 0.0,E5 0.0,E6 0.0}
DECL FDAT FSWP_60_9302={TOOL_NO 3,BASE_NO 3,IPO_FRAME #BASE,POINT2[] " "}
DECL LDAT LL_OLP80={VEL 2.0,ACC 100.0,APO_DIST 0.0,APO_FAC 0.0,ORI_TYP #VAR,CIRC_TYP #BASE,JERK_FAC 50.0}
DECL E6POS XSWP_60_9304={X 124.171097,Y 792.095215,Z 620.319885,A 159.417404,B 82.8863602,C 161.792404,S 18,T 42,E1 0.0,E2 0.0,E3 0.0,E4 0.0,E5 0.0,E6 0.0}
DECL FDAT FSWP_60_9304={TOOL_NO 3,BASE_NO 3,IPO_FRAME #BASE,POINT2[] " "}
DECL LDAT LL_OLP81={VEL 2.0,ACC 100.0,APO_DIST 0.0,APO_FAC 0.0,ORI_TYP #VAR,CIRC_TYP #BASE,JERK_FAC 50.0}
DECL E6POS XSWP_60_9306={X 132.870697,Y 841.648804,Z 621.361816,A 159.395203,B 82.8851624,C 161.773804,S 18,T 42,E1 0.0,E2 0.0,E3 0.0,E4 0.0,E5 0.0,E6 0.0}
DECL FDAT FSWP_60_9306={TOOL_NO 3,BASE_NO 3,IPO_FRAME #BASE,POINT2[] " "}
DECL LDAT LL_OLP82={VEL 2.0,ACC 100.0,APO_DIST 0.0,APO_FAC 0.0,ORI_TYP #VAR,CIRC_TYP #BASE,JERK_FAC 50.0}
DECL E6POS XSWP_60_9322={X 139.9673,Y 879.15332,Z 621.591309,A 159.403,B 82.8970566,C 167.299698,S 18,T 42,E1 0.0,E2 0.0,E3 0.0,E4 0.0,E5 0.0,E6 0.0}
DECL FDAT FSWP_60_9322={TOOL_NO 3,BASE_NO 3,IPO_FRAME #BASE,POINT2[] " "}
DECL E6POS Xl051={X 137.945007,Y 854.049988,Z 676.479004,A 164.794098,B 79.9898987,C 167.113907,S 2,T 42,E1 0.0,E2 0.0,E3 0.0,E4 0.0,E5 0.0,E6 0.0}
DECL FDAT Fl051={TOOL_NO 3,BASE_NO 3,IPO_FRAME #BASE,POINT2[] " "}
DECL E6POS XP5={X 420.465912,Y 747.624695,Z 1123.48804,A 158.533401,B 32.2998009,C 165.156693,S 18,T 42,E1 0.0,E2 0.0,E3 0.0,E4 0.0,E5 0.0,E6 0.0}
DECL FDAT FP5={TOOL_NO 3,BASE_NO 3,IPO_FRAME #BASE,POINT2[] " ",TQ_STATE FALSE}
DECL LDAT LCPDAT5={VEL 2.0,ACC 100.0,APO_DIST 10.0,APO_FAC 50.0,AXIS_VEL 100.0,AXIS_ACC 100.0,ORI_TYP #VAR,CIRC_TYP #BASE,JERK_FAC 50.0,GEAR_JERK 50.0,EXAX_IGN 0}
DECL E6POS XP6={X 1011.94702,Y 1316.37695,Z 872.489502,A -166.842194,B -74.2261429,C 77.8371201,S 18,T 34,E1 0.0,E2 0.0,E3 0.0,E4 0.0,E5 0.0,E6 0.0}
DECL FDAT FP6={TOOL_NO 3,BASE_NO 3,IPO_FRAME #BASE,POINT2[] " ",TQ_STATE FALSE}
DECL LDAT LL_OLP83={VEL 2.0,ACC 100.0,APO_DIST 2.0,APO_FAC 0.0,ORI_TYP #VAR,CIRC_TYP #BASE,JERK_FAC 50.0}
DECL E6POS Xl023={X 699.365295,Y 978.134216,Z 1321.15503,A -20.2005806,B -78.3323669,C -68.1035538,S 18,T 34,E1 0.0,E2 0.0,E3 0.0,E4 0.0,E5 0.0,E6 0.0}
DECL FDAT Fl023={TOOL_NO 3,BASE_NO 3,IPO_FRAME #BASE,POINT2[] " "}
DECL LDAT LL_OLP84={VEL 2.0,ACC 100.0,APO_DIST 0.0,APO_FAC 0.0,ORI_TYP #VAR,CIRC_TYP #BASE,JERK_FAC 50.0}
DECL LDAT LL_OLP85={VEL 2.0,ACC 100.0,APO_DIST 0.0,APO_FAC 0.0,ORI_TYP #VAR,CIRC_TYP #BASE,JERK_FAC 50.0}

DECL LDAT LL_OLP86={VEL 2.0,ACC 100.0,APO_DIST 0.0,APO_FAC 0.0,ORI_TYP #VAR,CIRC_TYP #BASE,JERK_FAC 50.0}

DECL LDAT LL_OLP87={VEL 2.0,ACC 100.0,APO_DIST 0.0,APO_FAC 0.0,ORI_TYP #VAR,CIRC_TYP #BASE,JERK_FAC 50.0}
DECL LDAT LL_OLP88={VEL 2.0,ACC 100.0,APO_DIST 0.0,APO_FAC 0.0,ORI_TYP #VAR,CIRC_TYP #BASE,JERK_FAC 50.0}
DECL LDAT LL_OLP89={VEL 2.0,ACC 100.0,APO_DIST 0.0,APO_FAC 0.0,ORI_TYP #VAR,CIRC_TYP #BASE,JERK_FAC 50.0}
DECL LDAT LL_OLP90={VEL 2.0,ACC 100.0,APO_DIST 0.0,APO_FAC 0.0,ORI_TYP #VAR,CIRC_TYP #BASE,JERK_FAC 50.0}
DECL LDAT LL_OLP91={VEL 2.0,ACC 100.0,APO_DIST 0.0,APO_FAC 0.0,ORI_TYP #VAR,CIRC_TYP #BASE,JERK_FAC 50.0}
DECL LDAT LL_OLP92={VEL 2.0,ACC 100.0,APO_DIST 0.0,APO_FAC 0.0,ORI_TYP #VAR,CIRC_TYP #BASE,JERK_FAC 50.0}
DECL LDAT LL_OLP93={VEL 2.0,ACC 100.0,APO_DIST 0.0,APO_FAC 0.0,ORI_TYP #VAR,CIRC_TYP #BASE,JERK_FAC 50.0}
DECL LDAT LL_OLP94={VEL 2.0,ACC 100.0,APO_DIST 0.0,APO_FAC 0.0,ORI_TYP #VAR,CIRC_TYP #BASE,JERK_FAC 50.0}
DECL E6POS Xl028={X 1184.32397,Y 978.322083,Z 1317.11304,A -14.4974499,B -74.4626236,C -73.6468124,S 18,T 34,E1 0.0,E2 0.0,E3 0.0,E4 0.0,E5 0.0,E6 0.0}


DECL FDAT Fl028={TOOL_NO 3,BASE_NO 3,IPO_FRAME #BASE,POINT2[] " "}
DECL LDAT LL_OLP95={VEL 2.0,ACC 100.0,APO_DIST 5.0,APO_FAC 0.0,ORI_TYP #VAR,CIRC_TYP #BASE,JERK_FAC 50.0}
DECL E6POS Xl033={X 1167.98999,Y 981.75531,Z 1261.08606,A -24.1799507,B -79.9280014,C -64.1580505,S 18,T 34,E1 0.0,E2 0.0,E3 0.0,E4 0.0,E5 0.0,E6 0.0}
DECL FDAT Fl033={TOOL_NO 3,BASE_NO 3,IPO_FRAME #BASE,POINT2[] " "}
DECL PDAT PPDAT1={VEL 100.0,ACC 100.0,APO_DIST 30.0,APO_MODE #CDIS,GEAR_JERK 50.0}
DECL E6POS XP7={X 1899.93604,Y 3567.76489,Z 589.863708,A -176.116592,B -26.2018795,C -91.7760925,S 18,T 42,E1 0.0,E2 0.0,E3 0.0,E4 0.0,E5 0.0,E6 0.0}

DECL FDAT FP7={TOOL_NO 4,BASE_NO 3,IPO_FRAME #BASE,POINT2[] " ",TQ_STATE FALSE}
DECL PDAT PPDAT2={VEL 100.0,ACC 100.0,APO_DIST 100.0,APO_MODE #CDIS,GEAR_JERK 50.0}
DECL LDAT LCPDAT7={VEL 2.0,ACC 100.0,APO_DIST 30.0,APO_FAC 50.0,AXIS_VEL 100.0,AXIS_ACC 100.0,ORI_TYP #VAR,CIRC_TYP #BASE,JERK_FAC 50.0,GEAR_JERK 50.0,EXAX_IGN 0}

DECL E6POS XSWP_60_8398={X 2127.00806,Y 1018.26501,Z 98.4453735,A 179.695496,B -26.7394199,C 91.8003998,S 18,T 34,E1 0.0,E2 0.0,E3 0.0,E4 0.0,E5 0.0,E6 0.0}
DECL FDAT FSWP_60_8398={TOOL_NO 3,BASE_NO 3,IPO_FRAME #BASE,POINT2[] " ",TQ_STATE FALSE}
DECL SPOT_SUGG_T LAST_SPOT={GUN[] " 1                      ",RETR_CMD[] "#OPN                    ",CHOISE[] "#FIRST                  ",CLO_TM[] "0                       ",PGNO1[] " 1                      ",PRESS1[] "0                       ",PGNO2[] " 1                      ",PRESS2[] "0                       ",SPOT_PARAMS[] "NORMAL                  "}
DECL SPOT_TYPE SNORMAL={GUN 1,PAIR #FIRST,RETR #OPN,CLO_TM 0,PGNO1 1,PRESS1 0.0,PGNO2 0,PRESS2 0.0}
DECL E6POS XSWP_60_9258={X 145.027603,Y 915.333679,Z 621.085388,A 92.0242233,B 54.5311508,C 101.880501,S 18,T 42,E1 0.0,E2 0.0,E3 0.0,E4 0.0,E5 0.0,E6 0.0}
DECL FDAT FSWP_60_9258={TOOL_NO 3,BASE_NO 3,IPO_FRAME #BASE,POINT2[] " ",TQ_STATE FALSE}
DECL LDAT LCPDAT6={VEL 2.0,ACC 100.0,APO_DIST 100.0,APO_FAC 50.0,AXIS_VEL 100.0,AXIS_ACC 100.0,ORI_TYP #VAR,CIRC_TYP #BASE,JERK_FAC 50.0,GEAR_JERK 50.0,EXAX_IGN 0}
DECL LDAT LCPDAT8={VEL 2.0,ACC 100.0,APO_DIST 10.0,APO_FAC 50.0,AXIS_VEL 100.0,AXIS_ACC 100.0,ORI_TYP #VAR,CIRC_TYP #BASE,JERK_FAC 50.0,GEAR_JERK 50.0,EXAX_IGN 0}
DECL LDAT LCPDAT9={VEL 2.0,ACC 100.0,APO_DIST 30.0,APO_FAC 50.0,AXIS_VEL 100.0,AXIS_ACC 100.0,ORI_TYP #VAR,CIRC_TYP #BASE,JERK_FAC 50.0,GEAR_JERK 50.0,EXAX_IGN 0}
DECL E6POS Xl066={X 1312.10205,Y 1148.0,Z 79.7080002,A 180.0,B -13.3133001,C 90.0,S 2,T 42}
DECL FDAT Fl066={TOOL_NO 3,BASE_NO 3,IPO_FRAME #BASE,POINT2[] " "}
DECL LDAT LCPDAT10={VEL 2.0,ACC 100.0,APO_DIST 5.0,APO_FAC 50.0,AXIS_VEL 100.0,AXIS_ACC 100.0,ORI_TYP #VAR,CIRC_TYP #BASE,JERK_FAC 50.0,GEAR_JERK 50.0,EXAX_IGN 0}
DECL E6POS XP4={X 1230.61096,Y 1015.41901,Z 62.1031799,A -179.999207,B -13.3151903,C 90.0011368,S 18,T 42,E1 0.0,E2 0.0,E3 0.0,E4 0.0,E5 0.0,E6 0.0}
DECL FDAT FP4={TOOL_NO 3,BASE_NO 3,IPO_FRAME #BASE,POINT2[] " ",TQ_STATE FALSE}
DECL LDAT LL_OLP27={VEL 2.0,ACC 100.0,APO_DIST 5.0,APO_FAC 0.0,ORI_TYP #VAR,CIRC_TYP #BASE,JERK_FAC 50.0}
DECL E6POS Xl071={X 1116.63403,Y 1017.16602,Z 51.4317093,A 179.996597,B -13.3109398,C 90.0032806,S 18,T 42,E1 0.0,E2 0.0,E3 0.0,E4 0.0,E5 0.0,E6 0.0}
DECL FDAT Fl071={TOOL_NO 3,BASE_NO 3,IPO_FRAME #BASE,POINT2[] " ",TQ_STATE FALSE}
DECL LDAT LCPDAT11={VEL 2.0,ACC 100.0,APO_DIST 5.0,APO_FAC 50.0,AXIS_VEL 100.0,AXIS_ACC 100.0,ORI_TYP #VAR,CIRC_TYP #BASE,JERK_FAC 50.0,GEAR_JERK 50.0,EXAX_IGN 0}
DECL E6POS XP8={X 1108.78296,Y 1017.35999,Z 73.2284927,A 179.996597,B -13.3102198,C 90.0024872,S 18,T 42,E1 0.0,E2 0.0,E3 0.0,E4 0.0,E5 0.0,E6 0.0}
DECL FDAT FP8={TOOL_NO 3,BASE_NO 3,IPO_FRAME #BASE,POINT2[] " ",TQ_STATE FALSE}
DECL LDAT LCPDAT12={VEL 2.0,ACC 100.0,APO_DIST 100.0,APO_FAC 50.0,AXIS_VEL 100.0,AXIS_ACC 100.0,ORI_TYP #VAR,CIRC_TYP #BASE,JERK_FAC 50.0,GEAR_JERK 50.0,EXAX_IGN 0}
DECL E6POS XSWP_61_7028={X 1103.71106,Y 1027.16394,Z 73.6532211,A 179.998795,B -13.3108597,C 90.0045013,S 18,T 42,E1 0.0,E2 0.0,E3 0.0,E4 0.0,E5 0.0,E6 0.0}
DECL FDAT FSWP_61_7028={TOOL_NO 3,BASE_NO 3,IPO_FRAME #BASE,POINT2[] " ",TQ_STATE FALSE}
DECL LDAT LCPDAT13={VEL 2.0,ACC 100.0,APO_DIST 100.0,APO_FAC 50.0,AXIS_VEL 100.0,AXIS_ACC 100.0,ORI_TYP #VAR,CIRC_TYP #BASE,JERK_FAC 50.0,GEAR_JERK 50.0,EXAX_IGN 0}
DECL E6POS XSWP_61_7030={X 1150.83301,Y 1025.60095,Z 92.6395035,A -179.999695,B -13.3080397,C 90.0064468,S 18,T 42,E1 0.0,E2 0.0,E3 0.0,E4 0.0,E5 0.0,E6 0.0}
DECL FDAT FSWP_61_7030={TOOL_NO 3,BASE_NO 3,IPO_FRAME #BASE,POINT2[] " ",TQ_STATE FALSE}
DECL LDAT LCPDAT14={VEL 2.0,ACC 100.0,APO_DIST 100.0,APO_FAC 50.0,AXIS_VEL 100.0,AXIS_ACC 100.0,ORI_TYP #VAR,CIRC_TYP #BASE,JERK_FAC 50.0,GEAR_JERK 50.0,EXAX_IGN 0}
DECL E6POS XSWP_61_7032={X 1207.69495,Y 1024.18103,Z 101.351501,A -179.906403,B -19.7679901,C 90.0272598,S 18,T 34,E1 0.0,E2 0.0,E3 0.0,E4 0.0,E5 0.0,E6 0.0}
DECL FDAT FSWP_61_7032={TOOL_NO 3,BASE_NO 3,IPO_FRAME #BASE,POINT2[] " ",TQ_STATE FALSE}
DECL LDAT LCPDAT15={VEL 2.0,ACC 100.0,APO_DIST 10.0,APO_FAC 50.0,AXIS_VEL 100.0,AXIS_ACC 100.0,ORI_TYP #VAR,CIRC_TYP #BASE,JERK_FAC 50.0,GEAR_JERK 50.0,EXAX_IGN 0}
DECL E6POS XP9={X 1206.38403,Y 1006.83502,Z 67.4408493,A -179.908997,B -19.7681408,C 90.0280304,S 18,T 34,E1 0.0,E2 0.0,E3 0.0,E4 0.0,E5 0.0,E6 0.0}
DECL FDAT FP9={TOOL_NO 3,BASE_NO 3,IPO_FRAME #BASE,POINT2[] " ",TQ_STATE FALSE}
DECL LDAT LCPDAT16={VEL 2.0,ACC 100.0,APO_DIST 10.0,APO_FAC 50.0,AXIS_VEL 100.0,AXIS_ACC 100.0,ORI_TYP #VAR,CIRC_TYP #BASE,JERK_FAC 50.0,GEAR_JERK 50.0,EXAX_IGN 0}
DECL E6POS XP10={X 1317.94104,Y 1023.60699,Z 57.3264008,A 179.9785,B -22.2589607,C 89.997467,S 18,T 34,E1 0.0,E2 0.0,E3 0.0,E4 0.0,E5 0.0,E6 0.0}
DECL FDAT FP10={TOOL_NO 3,BASE_NO 3,IPO_FRAME #BASE,POINT2[] " ",TQ_STATE FALSE}
DECL PDAT PPDAT3={VEL 100.0,ACC 100.0,APO_DIST 100.0,APO_MODE #CDIS,GEAR_JERK 50.0}
DECL PDAT PPDAT4={VEL 100.0,ACC 100.0,APO_DIST 100.0,APO_MODE #CDIS,GEAR_JERK 50.0}
ENDDAT
